  LIN {X 12250.007,Y 1961.237,Z 18.185,A 87.94718,B 0.00000,C 180.00000} ; preinsert
  LIN {X 12250.007,Y 1961.237,Z -231.815,A 87.94718,B 0.00000,C 180.00000} ; insert
  LIN {X 12250.007,Y 1961.237,Z -231.815,A 87.94718,B 0.00000,C 180.00000} ; release
  LIN {X 12250.007,Y 1961.237,Z 68.185,A 87.94718,B 0.00000,C 180.00000} ; retreat
  ; Step 908, bar 2215
  LIN {X 12850.007,Y 1961.237,Z 950.053,A 87.94718,B 0.00000,C 180.00000} ; outside
  LIN {X 12850.007,Y 1961.237,Z 18.185,A 87.94718,B 0.00000,C 180.00000} ; preinsert
  LIN {X 12850.007,Y 1961.237,Z -231.815,A 87.94718,B 0.00000,C 180.00000} ; insert
  LIN {X 12850.007,Y 1961.237,Z -231.815,A 87.94718,B 0.00000,C 180.00000} ; release
  LIN {X 12850.007,Y 1961.237,Z 68.185,A 87.94718,B 0.00000,C 180.00000} ; retreat
  ; Step 909, bar 2221
  LIN {X 13450.007,Y 1961.237,Z 950.053,A 87.94718,B 0.00000,C 180.00000} ; outside
  LIN {X 13450.007,Y 1961.237,Z 18.185,A 87.94718,B 0.00000,C 180.00000} ; preinsert
  LIN {X 13450.007,Y 1961.237,Z -231.815,A 87.94718,B 0.00000,C 180.00000} ; insert
  LIN {X 13450.007,Y 1961.237,Z -231.815,A 87.94718,B 0.00000,C 180.00000} ; release
  LIN {X 13450.007,Y 1961.237,Z 68.185,A 87.94718,B 0.00000,C 180.00000} ; retreat
  ; Step 910, bar 2227
  LIN {X 14050.007,Y 1961.237,Z 950.053,A 87.94718,B 0.00000,C 180.00000} ; outside
  LIN {X 14050.007,Y 1961.237,Z 18.185,A 87.94718,B 0.00000,C 180.00000} ; preinsert
  LIN {X 14050.007,Y 1961.237,Z -231.815,A 87.94718,B 0.00000,C 180.00000} ; insert
  LIN {X 14050.007,Y 1961.237,Z -231.815,A 87.94718,B 0.00000,C 180.00000} ; release
  LIN {X 14050.007,Y 1961.237,Z 68.185,A 87.94718,B 0.00000,C 180.00000} ; retreat
  ; Step 911, bar 2233
  LIN {X 14650.007,Y 1961.237,Z 950.053,A 87.94718,B 0.00000,C 180.00000} ; outside
  LIN {X 14650.007,Y 1961.237,Z 18.185,A 87.94718,B 0.00000,C 180.00000} ; preinsert
  LIN {X 14650.007,Y 1961.237,Z -231.815,A 87.94718,B 0.00000,C 180.00000} ; insert
  LIN {X 14650.007,Y 1961.237,Z -231.815,A 87.94718,B 0.00000,C 180.00000} ; release
  LIN {X 14650.007,Y 1961.237,Z 68.185,A 87.94718,B 0.00000,C 180.00000} ; retreat
  ; Step 912, bar 2239
  LIN {X 15250.007,Y 1961.237,Z 950.053,A 87.94718,B 0.00000,C 180.00000} ; outside
  LIN {X 15250.007,Y 1961.237,Z 18.185,A 87.94718,B 0.00000,C 180.00000} ; preinsert
  LIN {X 15250.007,Y 1961.237,Z -231.815,A 87.94718,B 0.00000,C 180.00000} ; insert
  LIN {X 15250.007,Y 1961.237,Z -231.815,A 87.94718,B 0.00000,C 180.00000} ; release
  LIN {X 15250.007,Y 1961.237,Z 68.185,A 87.94718,B 0.00000,C 180.00000} ; retreat
  ; Step 913, bar 2245
  LIN {X 15850.007,Y 1961.237,Z 950.053,A 87.94718,B 0.00000,C 180.00000} ; outside
  LIN {X 15850.007,Y 1961.237,Z 18.185,A 87.94718,B 0.00000,C 180.00000} ; preinsert
  LIN {X 15850.007,Y 1961.237,Z -231.815,A 87.94718,B 0.00000,C 180.00000} ; insert
  LIN {X 15850.007,Y 1961.237,Z -231.815,A 87.94718,B 0.00000,C 180.00000} ; release
  LIN {X 15850.007,Y 1961.237,Z 68.185,A 87.94718,B 0.00000,C 180.00000} ; retreat
  ; Step 914, bar 298
  LIN {X 0.000,Y -2740.000,Z 1104.371,A 0.00000,B 0.00000,C 180.00000} ; outside
  LIN {X 0.000,Y -2740.000,Z 176.496,A 0.00000,B 0.00000,C 180.00000} ; preinsert
  LIN {X 0.000,Y -2740.000,Z -73.504,A 0.00000,B 0.00000,C 180.00000} ; insert
  LIN {X 0.000,Y -2740.000,Z -73.504,A 0.00000,B 0.00000,C 180.00000} ; release
  LIN {X 0.000,Y -2740.000,Z 226.496,A 0.00000,B 0.00000,C 180.00000} ; retreat
  ; Step 915, bar 325
  LIN {X 0.000,Y 2740.000,Z 1104.371,A 0.00000,B 0.00000,C 180.00000} ; outside
  LIN {X 0.000,Y 2740.000,Z 176.496,A 0.00000,B 0.00000,C 180.00000} ; preinsert
  LIN {X 0.000,Y 2740.000,Z -73.504,A 0.00000,B 0.00000,C 180.00000} ; insert
  LIN {X 0.000,Y 2740.000,Z -73.504,A 0.00000,B 0.00000,C 180.00000} ; release
  LIN {X 0.000,Y 2740.000,Z 226.496,A 0.00000,B 0.00000,C 180.00000} ; retreat
  ; Step 916, bar 284
  LIN {X 0.000,Y -750.000,Z 1108.746,A 0.00000,B 0.00000,C 180.00000} ; outside
  LIN {X 0.000,Y -750.000,Z 178.683,A 0.00000,B 0.00000,C 180.00000} ; preinsert
  LIN {X 0.000,Y -750.000,Z -71.317,A 0.00000,B 0.00000,C 180.00000} ; insert
  LIN {X 0.000,Y -750.000,Z -71.317,A 0.00000,B 0.00000,C 180.00000} ; release
  LIN {X 0.000,Y -750.000,Z 228.683,A 0.00000,B 0.00000,C 180.00000} ; retreat
  ; Step 917, bar 311
  LIN {X 0.000,Y 750.000,Z 1108.746,A 0.00000,B 0.00000,C 180.00000} ; outside
  LIN {X 0.000,Y 750.000,Z 178.683,A 0.00000,B 0.00000,C 180.00000} ; preinsert
  LIN {X 0.000,Y 750.000,Z -71.317,A 0.00000,B 0.00000,C 180.00000} ; insert
  LIN {X 0.000,Y 750.000,Z -71.317,A 0.00000,B 0.00000,C 180.00000} ; release
  LIN {X 0.000,Y 750.000,Z 228.683,A 0.00000,B 0.00000,C 180.00000} ; retreat
  ; Step 918, bar 3105
  LIN {X -15204.133,Y -641.217,Z 1079.276,A -179.87076,B 0.00000,C 180.00000} ; outside
  LIN {X -15204.133,Y -641.217,Z 104.517,A -179.87076,B 0.00000,C 180.00000} ; preinsert
  LIN {X -15204.133,Y -641.217,Z -145.483,A -179.87076,B 0.00000,C 180.00000} ; insert
  LIN {X -15204.133,Y -641.217,Z -145.483,A -179.87076,B 0.00000,C 180.00000} ; release
  LIN {X -15204.133,Y -641.217,Z 154.517,A -179.87076,B 0.00000,C 180.00000} ; retreat
  ; Step 919, bar 3095
  LIN {X 15204.133,Y -641.217,Z 1079.276,A -0.12924,B 0.00000,C 180.00000} ; outside
  LIN {X 15204.133,Y -641.217,Z 104.517,A -0.12924,B 0.00000,C 180.00000} ; preinsert
  LIN {X 15204.133,Y -641.217,Z -145.483,A -0.12924,B 0.00000,C 180.00000} ; insert
  LIN {X 15204.133,Y -641.217,Z -145.483,A -0.12924,B 0.00000,C 180.00000} ; release
  LIN {X 15204.133,Y -641.217,Z 154.517,A -0.12924,B 0.00000,C 180.00000} ; retreat
  ; Step 920, bar 3100
  LIN {X -15204.133,Y 641.217,Z 1079.276,A 179.87076,B 0.00000,C 180.00000} ; outside
  LIN {X -15204.133,Y 641.217,Z 104.517,A 179.87076,B 0.00000,C 180.00000} ; preinsert
  LIN {X -15204.133,Y 641.217,Z -145.483,A 179.87076,B 0.00000,C 180.00000} ; insert
  LIN {X -15204.133,Y 641.217,Z -145.483,A 179.87076,B 0.00000,C 180.00000} ; release
  LIN {X -15204.133,Y 641.217,Z 154.517,A 179.87076,B 0.00000,C 180.00000} ; retreat
  ; Step 921, bar 3090
  LIN {X 15204.133,Y 641.217,Z 1079.276,A 0.12924,B 0.00000,C 180.00000} ; outside
  LIN {X 15204.133,Y 641.217,Z 104.517,A 0.12924,B 0.00000,C 180.00000} ; preinsert
  LIN {X 15204.133,Y 641.217,Z -145.483,A 0.12924,B 0.00000,C 180.00000} ; insert
  LIN {X 15204.133,Y 641.217,Z -145.483,A 0.12924,B 0.00000,C 180.00000} ; release
  LIN {X 15204.133,Y 641.217,Z 154.517,A 0.12924,B 0.00000,C 180.00000} ; retreat
  ; Step 922, bar 2755
  LIN {X -1500.007,Y -1396.237,Z 955.597,A -92.05282,B 0.00000,C -180.00000} ; outside
  LIN {X -1500.007,Y -1396.237,Z 24.092,A -92.05282,B 0.00000,C -180.00000} ; preinsert
  LIN {X -1500.007,Y -1396.237,Z -225.908,A -92.05282,B 0.00000,C -180.00000} ; insert
  LIN {X -1500.007,Y -1396.237,Z -225.908,A -92.05282,B 0.00000,C -180.00000} ; release
  LIN {X -1500.007,Y -1396.237,Z 74.092,A -92.05282,B 0.00000,C -180.00000} ; retreat
  ; Step 923, bar 2752
  LIN {X -750.007,Y -1396.237,Z 955.597,A -92.05282,B 0.00000,C -180.00000} ; outside
  LIN {X -750.007,Y -1396.237,Z 24.092,A -92.05282,B 0.00000,C -180.00000} ; preinsert
  LIN {X -750.007,Y -1396.237,Z -225.908,A -92.05282,B 0.00000,C -180.00000} ; insert
  LIN {X -750.007,Y -1396.237,Z -225.908,A -92.05282,B 0.00000,C -180.00000} ; release
  LIN {X -750.007,Y -1396.237,Z 74.092,A -92.05282,B 0.00000,C -180.00000} ; retreat
  ; Step 924, bar 2749
  LIN {X -0.007,Y -1396.237,Z 955.597,A -92.05282,B 0.00000,C -180.00000} ; outside
  LIN {X -0.007,Y -1396.237,Z 24.092,A -92.05282,B 0.00000,C -180.00000} ; preinsert
  LIN {X -0.007,Y -1396.237,Z -225.908,A -92.05282,B 0.00000,C -180.00000} ; insert
  LIN {X -0.007,Y -1396.237,Z -225.908,A -92.05282,B 0.00000,C -180.00000} ; release
  LIN {X -0.007,Y -1396.237,Z 74.092,A -92.05282,B 0.00000,C -180.00000} ; retreat
  ; Step 925, bar 2758
  LIN {X -2250.007,Y -1396.237,Z 955.597,A -92.05282,B 0.00000,C -180.00000} ; outside
  LIN {X -2250.007,Y -1396.237,Z 24.092,A -92.05282,B 0.00000,C -180.00000} ; preinsert
  LIN {X -2250.007,Y -1396.237,Z -225.908,A -92.05282,B 0.00000,C -180.00000} ; insert
  LIN {X -2250.007,Y -1396.237,Z -225.908,A -92.05282,B 0.00000,C -180.00000} ; release
  LIN {X -2250.007,Y -1396.237,Z 74.092,A -92.05282,B 0.00000,C -180.00000} ; retreat
  ; Step 926, bar 2761
  LIN {X -3000.007,Y -1396.237,Z 955.597,A -92.05282,B 0.00000,C -180.00000} ; outside
  LIN {X -3000.007,Y -1396.237,Z 24.092,A -92.05282,B 0.00000,C -180.00000} ; preinsert
  LIN {X -3000.007,Y -1396.237,Z -225.908,A -92.05282,B 0.00000,C -180.00000} ; insert
  LIN {X -3000.007,Y -1396.237,Z -225.908,A -92.05282,B 0.00000,C -180.00000} ; release
  LIN {X -3000.007,Y -1396.237,Z 74.092,A -92.05282,B 0.00000,C -180.00000} ; retreat
  ; Step 927, bar 2764
  LIN {X -3750.007,Y -1396.237,Z 955.597,A -92.05282,B 0.00000,C -180.00000} ; outside
  LIN {X -3750.007,Y -1396.237,Z 24.092,A -92.05282,B 0.00000,C -180.00000} ; preinsert
  LIN {X -3750.007,Y -1396.237,Z -225.908,A -92.05282,B 0.00000,C -180.00000} ; insert
  LIN {X -3750.007,Y -1396.237,Z -225.908,A -92.05282,B 0.00000,C -180.00000} ; release
  LIN {X -3750.007,Y -1396.237,Z 74.092,A -92.05282,B 0.00000,C -180.00000} ; retreat
  ; Step 928, bar 2767
  LIN {X -4500.007,Y -1396.237,Z 955.597,A -92.05282,B 0.00000,C -180.00000} ; outside
  LIN {X -4500.007,Y -1396.237,Z 24.092,A -92.05282,B 0.00000,C -180.00000} ; preinsert
  LIN {X -4500.007,Y -1396.237,Z -225.908,A -92.05282,B 0.00000,C -180.00000} ; insert
  LIN {X -4500.007,Y -1396.237,Z -225.908,A -92.05282,B 0.00000,C -180.00000} ; release
  LIN {X -4500.007,Y -1396.237,Z 74.092,A -92.05282,B 0.00000,C -180.00000} ; retreat
  ; Step 929, bar 2770
  LIN {X -5250.007,Y -1396.237,Z 955.597,A -92.05282,B 0.00000,C -180.00000} ; outside
  LIN {X -5250.007,Y -1396.237,Z 24.092,A -92.05282,B 0.00000,C -180.00000} ; preinsert
  LIN {X -5250.007,Y -1396.237,Z -225.908,A -92.05282,B 0.00000,C -180.00000} ; insert
  LIN {X -5250.007,Y -1396.237,Z -225.908,A -92.05282,B 0.00000,C -180.00000} ; release
  LIN {X -5250.007,Y -1396.237,Z 74.092,A -92.05282,B 0.00000,C -180.00000} ; retreat
  ; Step 930, bar 2773
  LIN {X -6000.007,Y -1396.237,Z 955.597,A -92.05282,B 0.00000,C -180.00000} ; outside
  LIN {X -6000.007,Y -1396.237,Z 24.092,A -92.05282,B 0.00000,C -180.00000} ; preinsert
  LIN {X -6000.007,Y -1396.237,Z -225.908,A -92.05282,B 0.00000,C -180.00000} ; insert
  LIN {X -6000.007,Y -1396.237,Z -225.908,A -92.05282,B 0.00000,C -180.00000} ; release
  LIN {X -6000.007,Y -1396.237,Z 74.092,A -92.05282,B 0.00000,C -180.00000} ; retreat
  ; Step 931, bar 2776
  LIN {X -6750.007,Y -1396.237,Z 955.597,A -92.05282,B 0.00000,C -180.00000} ; outside
  LIN {X -6750.007,Y -1396.237,Z 24.092,A -92.05282,B 0.00000,C -180.00000} ; preinsert
  LIN {X -6750.007,Y -1396.237,Z -225.908,A -92.05282,B 0.00000,C -180.00000} ; insert
  LIN {X -6750.007,Y -1396.237,Z -225.908,A -92.05282,B 0.00000,C -180.00000} ; release
  LIN {X -6750.007,Y -1396.237,Z 74.092,A -92.05282,B 0.00000,C -180.00000} ; retreat
  ; Step 932, bar 2779
  LIN {X -7500.007,Y -1396.237,Z 955.597,A -92.05282,B 0.00000,C -180.00000} ; outside
  LIN {X -7500.007,Y -1396.237,Z 24.092,A -92.05282,B 0.00000,C -180.00000} ; preinsert
  LIN {X -7500.007,Y -1396.237,Z -225.908,A -92.05282,B 0.00000,C -180.00000} ; insert
  LIN {X -7500.007,Y -1396.237,Z -225.908,A -92.05282,B 0.00000,C -180.00000} ; release
  LIN {X -7500.007,Y -1396.237,Z 74.092,A -92.05282,B 0.00000,C -180.00000} ; retreat
  ; Step 933, bar 2782
  LIN {X -8250.007,Y -1396.237,Z 955.597,A -92.05282,B 0.00000,C -180.00000} ; outside
  LIN {X -8250.007,Y -1396.237,Z 24.092,A -92.05282,B 0.00000,C -180.00000} ; preinsert
  LIN {X -8250.007,Y -1396.237,Z -225.908,A -92.05282,B 0.00000,C -180.00000} ; insert
  LIN {X -8250.007,Y -1396.237,Z -225.908,A -92.05282,B 0.00000,C -180.00000} ; release
  LIN {X -8250.007,Y -1396.237,Z 74.092,A -92.05282,B 0.00000,C -180.00000} ; retreat
  ; Step 934, bar 2785
  LIN {X -9000.007,Y -1396.237,Z 955.597,A -92.05282,B 0.00000,C -180.00000} ; outside
  LIN {X -9000.007,Y -1396.237,Z 24.092,A -92.05282,B 0.00000,C -180.00000} ; preinsert
  LIN {X -9000.007,Y -1396.237,Z -225.908,A -92.05282,B 0.00000,C -180.00000} ; insert
  LIN {X -9000.007,Y -1396.237,Z -225.908,A -92.05282,B 0.00000,C -180.00000} ; release
  LIN {X -9000.007,Y -1396.237,Z 74.092,A -92.05282,B 0.00000,C -180.00000} ; retreat
  ; Step 935, bar 2788
  LIN {X -9750.007,Y -1396.237,Z 955.597,A -92.05282,B 0.00000,C -180.00000} ; outside
  LIN {X -9750.007,Y -1396.237,Z 24.092,A -92.05282,B 0.00000,C -180.00000} ; preinsert
  LIN {X -9750.007,Y -1396.237,Z -225.908,A -92.05282,B 0.00000,C -180.00000} ; insert
  LIN {X -9750.007,Y -1396.237,Z -225.908,A -92.05282,B 0.00000,C -180.00000} ; release
  LIN {X -9750.007,Y -1396.237,Z 74.092,A -92.05282,B 0.00000,C -180.00000} ; retreat
  ; Step 936, bar 2791
  LIN {X -10500.007,Y -1396.237,Z 955.597,A -92.05282,B 0.00000,C -180.00000} ; outside
  LIN {X -10500.007,Y -1396.237,Z 24.092,A -92.05282,B 0.00000,C -180.00000} ; preinsert
  LIN {X -10500.007,Y -1396.237,Z -225.908,A -92.05282,B 0.00000,C -180.00000} ; insert
  LIN {X -10500.007,Y -1396.237,Z -225.908,A -92.05282,B 0.00000,C -180.00000} ; release
  LIN {X -10500.007,Y -1396.237,Z 74.092,A -92.05282,B 0.00000,C -180.00000} ; retreat
  ; Step 937, bar 2794
  LIN {X -11250.007,Y -1396.237,Z 955.597,A -92.05282,B 0.00000,C -180.00000} ; outside
  LIN {X -11250.007,Y -1396.237,Z 24.092,A -92.05282,B 0.00000,C -180.00000} ; preinsert
  LIN {X -11250.007,Y -1396.237,Z -225.908,A -92.05282,B 0.00000,C -180.00000} ; insert
  LIN {X -11250.007,Y -1396.237,Z -225.908,A -92.05282,B 0.00000,C -180.00000} ; release
  LIN {X -11250.007,Y -1396.237,Z 74.092,A -92.05282,B 0.00000,C -180.00000} ; retreat
  ; Step 938, bar 2797
  LIN {X -12000.007,Y -1396.237,Z 955.597,A -92.05282,B 0.00000,C -180.00000} ; outside
  LIN {X -12000.007,Y -1396.237,Z 24.092,A -92.05282,B 0.00000,C -180.00000} ; preinsert
  LIN {X -12000.007,Y -1396.237,Z -225.908,A -92.05282,B 0.00000,C -180.00000} ; insert
  LIN {X -12000.007,Y -1396.237,Z -225.908,A -92.05282,B 0.00000,C -180.00000} ; release
  LIN {X -12000.007,Y -1396.237,Z 74.092,A -92.05282,B 0.00000,C -180.00000} ; retreat
  ; Step 939, bar 2638
  LIN {X 750.007,Y 1396.237,Z 955.597,A 87.94718,B 0.00000,C 180.00000} ; outside
  LIN {X 750.007,Y 1396.237,Z 24.092,A 87.94718,B 0.00000,C 180.00000} ; preinsert
  LIN {X 750.007,Y 1396.237,Z -225.908,A 87.94718,B 0.00000,C 180.00000} ; insert
  LIN {X 750.007,Y 1396.237,Z -225.908,A 87.94718,B 0.00000,C 180.00000} ; release
  LIN {X 750.007,Y 1396.237,Z 74.092,A 87.94718,B 0.00000,C 180.00000} ; retreat
  ; Step 940, bar 2641
  LIN {X 1500.007,Y 1396.237,Z 955.597,A 87.94718,B 0.00000,C -180.00000} ; outside
  LIN {X 1500.007,Y 1396.237,Z 24.092,A 87.94718,B 0.00000,C -180.00000} ; preinsert
  LIN {X 1500.007,Y 1396.237,Z -225.908,A 87.94718,B 0.00000,C -180.00000} ; insert
  LIN {X 1500.007,Y 1396.237,Z -225.908,A 87.94718,B 0.00000,C -180.00000} ; release
  LIN {X 1500.007,Y 1396.237,Z 74.092,A 87.94718,B 0.00000,C -180.00000} ; retreat
  ; Step 941, bar 2644
  LIN {X 2250.007,Y 1396.237,Z 955.597,A 87.94718,B 0.00000,C -180.00000} ; outside
  LIN {X 2250.007,Y 1396.237,Z 24.092,A 87.94718,B 0.00000,C -180.00000} ; preinsert
  LIN {X 2250.007,Y 1396.237,Z -225.908,A 87.94718,B 0.00000,C -180.00000} ; insert
  LIN {X 2250.007,Y 1396.237,Z -225.908,A 87.94718,B 0.00000,C -180.00000} ; release
  LIN {X 2250.007,Y 1396.237,Z 74.092,A 87.94718,B 0.00000,C -180.00000} ; retreat
  ; Step 942, bar 2647
  LIN {X 3000.007,Y 1396.237,Z 955.597,A 87.94718,B 0.00000,C -180.00000} ; outside
  LIN {X 3000.007,Y 1396.237,Z 24.092,A 87.94718,B 0.00000,C -180.00000} ; preinsert
  LIN {X 3000.007,Y 1396.237,Z -225.908,A 87.94718,B 0.00000,C -180.00000} ; insert
  LIN {X 3000.007,Y 1396.237,Z -225.908,A 87.94718,B 0.00000,C -180.00000} ; release
  LIN {X 3000.007,Y 1396.237,Z 74.092,A 87.94718,B 0.00000,C -180.00000} ; retreat
  ; Step 943, bar 2650
  LIN {X 3750.007,Y 1396.237,Z 955.597,A 87.94718,B 0.00000,C -180.00000} ; outside
  LIN {X 3750.007,Y 1396.237,Z 24.092,A 87.94718,B 0.00000,C -180.00000} ; preinsert
  LIN {X 3750.007,Y 1396.237,Z -225.908,A 87.94718,B 0.00000,C -180.00000} ; insert
  LIN {X 3750.007,Y 1396.237,Z -225.908,A 87.94718,B 0.00000,C -180.00000} ; release
  LIN {X 3750.007,Y 1396.237,Z 74.092,A 87.94718,B 0.00000,C -180.00000} ; retreat
  ; Step 944, bar 2653
  LIN {X 4500.007,Y 1396.237,Z 955.597,A 87.94718,B 0.00000,C 180.00000} ; outside
  LIN {X 4500.007,Y 1396.237,Z 24.092,A 87.94718,B 0.00000,C 180.00000} ; preinsert
  LIN {X 4500.007,Y 1396.237,Z -225.908,A 87.94718,B 0.00000,C 180.00000} ; insert
  LIN {X 4500.007,Y 1396.237,Z -225.908,A 87.94718,B 0.00000,C 180.00000} ; release
  LIN {X 4500.007,Y 1396.237,Z 74.092,A 87.94718,B 0.00000,C 180.00000} ; retreat
  ; Step 945, bar 2656
  LIN {X 5250.007,Y 1396.237,Z 955.597,A 87.94718,B 0.00000,C 180.00000} ; outside
  LIN {X 5250.007,Y 1396.237,Z 24.092,A 87.94718,B 0.00000,C 180.00000} ; preinsert
  LIN {X 5250.007,Y 1396.237,Z -225.908,A 87.94718,B 0.00000,C 180.00000} ; insert
  LIN {X 5250.007,Y 1396.237,Z -225.908,A 87.94718,B 0.00000,C 180.00000} ; release
  LIN {X 5250.007,Y 1396.237,Z 74.092,A 87.94718,B 0.00000,C 180.00000} ; retreat
  ; Step 946, bar 2659
  LIN {X 6000.007,Y 1396.237,Z 955.597,A 87.94718,B 0.00000,C 180.00000} ; outside
  LIN {X 6000.007,Y 1396.237,Z 24.092,A 87.94718,B 0.00000,C 180.00000} ; preinsert
  LIN {X 6000.007,Y 1396.237,Z -225.908,A 87.94718,B 0.00000,C 180.00000} ; insert
  LIN {X 6000.007,Y 1396.237,Z -225.908,A 87.94718,B 0.00000,C 180.00000} ; release
  LIN {X 6000.007,Y 1396.237,Z 74.092,A 87.94718,B 0.00000,C 180.00000} ; retreat
  ; Step 947, bar 2662
  LIN {X 6750.007,Y 1396.237,Z 955.597,A 87.94718,B 0.00000,C 180.00000} ; outside
  LIN {X 6750.007,Y 1396.237,Z 24.092,A 87.94718,B 0.00000,C 180.00000} ; preinsert
  LIN {X 6750.007,Y 1396.237,Z -225.908,A 87.94718,B 0.00000,C 180.00000} ; insert
  LIN {X 6750.007,Y 1396.237,Z -225.908,A 87.94718,B 0.00000,C 180.00000} ; release
  LIN {X 6750.007,Y 1396.237,Z 74.092,A 87.94718,B 0.00000,C 180.00000} ; retreat
  ; Step 948, bar 2665
  LIN {X 7500.007,Y 1396.237,Z 955.597,A 87.94718,B 0.00000,C 180.00000} ; outside
  LIN {X 7500.007,Y 1396.237,Z 24.092,A 87.94718,B 0.00000,C 180.00000} ; preinsert
  LIN {X 7500.007,Y 1396.237,Z -225.908,A 87.94718,B 0.00000,C 180.00000} ; insert
  LIN {X 7500.007,Y 1396.237,Z -225.908,A 87.94718,B 0.00000,C 180.00000} ; release
  LIN {X 7500.007,Y 1396.237,Z 74.092,A 87.94718,B 0.00000,C 180.00000} ; retreat
  ; Step 949, bar 2668
  LIN {X 8250.007,Y 1396.237,Z 955.597,A 87.94718,B 0.00000,C 180.00000} ; outside
  LIN {X 8250.007,Y 1396.237,Z 24.092,A 87.94718,B 0.00000,C 180.00000} ; preinsert
  LIN {X 8250.007,Y 1396.237,Z -225.908,A 87.94718,B 0.00000,C 180.00000} ; insert
  LIN {X 8250.007,Y 1396.237,Z -225.908,A 87.94718,B 0.00000,C 180.00000} ; release
  LIN {X 8250.007,Y 1396.237,Z 74.092,A 87.94718,B 0.00000,C 180.00000} ; retreat
  ; Step 950, bar 2671
  LIN {X 9000.007,Y 1396.237,Z 955.597,A 87.94718,B 0.00000,C 180.00000} ; outside
  LIN {X 9000.007,Y 1396.237,Z 24.092,A 87.94718,B 0.00000,C 180.00000} ; preinsert
  LIN {X 9000.007,Y 1396.237,Z -225.908,A 87.94718,B 0.00000,C 180.00000} ; insert
  LIN {X 9000.007,Y 1396.237,Z -225.908,A 87.94718,B 0.00000,C 180.00000} ; release
  LIN {X 9000.007,Y 1396.237,Z 74.092,A 87.94718,B 0.00000,C 180.00000} ; retreat
  ; Step 951, bar 2674
  LIN {X 9750.007,Y 1396.237,Z 955.597,A 87.94718,B 0.00000,C 180.00000} ; outside
  LIN {X 9750.007,Y 1396.237,Z 24.092,A 87.94718,B 0.00000,C 180.00000} ; preinsert
  LIN {X 9750.007,Y 1396.237,Z -225.908,A 87.94718,B 0.00000,C 180.00000} ; insert
  LIN {X 9750.007,Y 1396.237,Z -225.908,A 87.94718,B 0.00000,C 180.00000} ; release
  LIN {X 9750.007,Y 1396.237,Z 74.092,A 87.94718,B 0.00000,C 180.00000} ; retreat
  ; Step 952, bar 2677
  LIN {X 10500.007,Y 1396.237,Z 955.597,A 87.94718,B 0.00000,C 180.00000} ; outside
  LIN {X 10500.007,Y 1396.237,Z 24.092,A 87.94718,B 0.00000,C 180.00000} ; preinsert
  LIN {X 10500.007,Y 1396.237,Z -225.908,A 87.94718,B 0.00000,C 180.00000} ; insert
  LIN {X 10500.007,Y 1396.237,Z -225.908,A 87.94718,B 0.00000,C 180.00000} ; release
  LIN {X 10500.007,Y 1396.237,Z 74.092,A 87.94718,B 0.00000,C 180.00000} ; retreat
  ; Step 953, bar 2680
  LIN {X 11250.007,Y 1396.237,Z 955.597,A 87.94718,B 0.00000,C 180.00000} ; outside
  LIN {X 11250.007,Y 1396.237,Z 24.092,A 87.94718,B 0.00000,C 180.00000} ; preinsert
  LIN {X 11250.007,Y 1396.237,Z -225.908,A 87.94718,B 0.00000,C 180.00000} ; insert
  LIN {X 11250.007,Y 1396.237,Z -225.908,A 87.94718,B 0.00000,C 180.00000} ; release
  LIN {X 11250.007,Y 1396.237,Z 74.092,A 87.94718,B 0.00000,C 180.00000} ; retreat
  ; Step 954, bar 2683
  LIN {X 12000.007,Y 1396.237,Z 955.597,A 87.94718,B 0.00000,C 180.00000} ; outside
  LIN {X 12000.007,Y 1396.237,Z 24.092,A 87.94718,B 0.00000,C 180.00000} ; preinsert
  LIN {X 12000.007,Y 1396.237,Z -225.908,A 87.94718,B 0.00000,C 180.00000} ; insert
  LIN {X 12000.007,Y 1396.237,Z -225.908,A 87.94718,B 0.00000,C 180.00000} ; release
  LIN {X 12000.007,Y 1396.237,Z 74.092,A 87.94718,B 0.00000,C 180.00000} ; retreat
  ; Step 955, bar 2800
  LIN {X 750.007,Y -1396.237,Z 955.597,A -87.94718,B 0.00000,C 180.00000} ; outside
  LIN {X 750.007,Y -1396.237,Z 24.092,A -87.94718,B 0.00000,C 180.00000} ; preinsert
  LIN {X 750.007,Y -1396.237,Z -225.908,A -87.94718,B 0.00000,C 180.00000} ; insert
  LIN {X 750.007,Y -1396.237,Z -225.908,A -87.94718,B 0.00000,C 180.00000} ; release
  LIN {X 750.007,Y -1396.237,Z 74.092,A -87.94718,B 0.00000,C 180.00000} ; retreat
  ; Step 956, bar 2803
  LIN {X 1500.007,Y -1396.237,Z 955.597,A -87.94718,B 0.00000,C -180.00000} ; outside
  LIN {X 1500.007,Y -1396.237,Z 24.092,A -87.94718,B 0.00000,C -180.00000} ; preinsert
  LIN {X 1500.007,Y -1396.237,Z -225.908,A -87.94718,B 0.00000,C -180.00000} ; insert
  LIN {X 1500.007,Y -1396.237,Z -225.908,A -87.94718,B 0.00000,C -180.00000} ; release
  LIN {X 1500.007,Y -1396.237,Z 74.092,A -87.94718,B 0.00000,C -180.00000} ; retreat
  ; Step 957, bar 2806
  LIN {X 2250.007,Y -1396.237,Z 955.597,A -87.94718,B 0.00000,C -180.00000} ; outside
  LIN {X 2250.007,Y -1396.237,Z 24.092,A -87.94718,B 0.00000,C -180.00000} ; preinsert
  LIN {X 2250.007,Y -1396.237,Z -225.908,A -87.94718,B 0.00000,C -180.00000} ; insert
  LIN {X 2250.007,Y -1396.237,Z -225.908,A -87.94718,B 0.00000,C -180.00000} ; release
  LIN {X 2250.007,Y -1396.237,Z 74.092,A -87.94718,B 0.00000,C -180.00000} ; retreat
  ; Step 958, bar 2809
  LIN {X 3000.007,Y -1396.237,Z 955.597,A -87.94718,B 0.00000,C -180.00000} ; outside
  LIN {X 3000.007,Y -1396.237,Z 24.092,A -87.94718,B 0.00000,C -180.00000} ; preinsert
  LIN {X 3000.007,Y -1396.237,Z -225.908,A -87.94718,B 0.00000,C -180.00000} ; insert
  LIN {X 3000.007,Y -1396.237,Z -225.908,A -87.94718,B 0.00000,C -180.00000} ; release
  LIN {X 3000.007,Y -1396.237,Z 74.092,A -87.94718,B 0.00000,C -180.00000} ; retreat
  ; Step 959, bar 2812
  LIN {X 3750.007,Y -1396.237,Z 955.597,A -87.94718,B 0.00000,C -180.00000} ; outside
  LIN {X 3750.007,Y -1396.237,Z 24.092,A -87.94718,B 0.00000,C -180.00000} ; preinsert
  LIN {X 3750.007,Y -1396.237,Z -225.908,A -87.94718,B 0.00000,C -180.00000} ; insert
  LIN {X 3750.007,Y -1396.237,Z -225.908,A -87.94718,B 0.00000,C -180.00000} ; release
  LIN {X 3750.007,Y -1396.237,Z 74.092,A -87.94718,B 0.00000,C -180.00000} ; retreat
  ; Step 960, bar 2815
  LIN {X 4500.007,Y -1396.237,Z 955.597,A -87.94718,B 0.00000,C 180.00000} ; outside
  LIN {X 4500.007,Y -1396.237,Z 24.092,A -87.94718,B 0.00000,C 180.00000} ; preinsert
  LIN {X 4500.007,Y -1396.237,Z -225.908,A -87.94718,B 0.00000,C 180.00000} ; insert
  LIN {X 4500.007,Y -1396.237,Z -225.908,A -87.94718,B 0.00000,C 180.00000} ; release
  LIN {X 4500.007,Y -1396.237,Z 74.092,A -87.94718,B 0.00000,C 180.00000} ; retreat
  ; Step 961, bar 2818
  LIN {X 5250.007,Y -1396.237,Z 955.597,A -87.94718,B 0.00000,C 180.00000} ; outside
  LIN {X 5250.007,Y -1396.237,Z 24.092,A -87.94718,B 0.00000,C 180.00000} ; preinsert
  LIN {X 5250.007,Y -1396.237,Z -225.908,A -87.94718,B 0.00000,C 180.00000} ; insert
  LIN {X 5250.007,Y -1396.237,Z -225.908,A -87.94718,B 0.00000,C 180.00000} ; release
  LIN {X 5250.007,Y -1396.237,Z 74.092,A -87.94718,B 0.00000,C 180.00000} ; retreat
  ; Step 962, bar 2821
  LIN {X 6000.007,Y -1396.237,Z 955.597,A -87.94718,B 0.00000,C 180.00000} ; outside
  LIN {X 6000.007,Y -1396.237,Z 24.092,A -87.94718,B 0.00000,C 180.00000} ; preinsert
  LIN {X 6000.007,Y -1396.237,Z -225.908,A -87.94718,B 0.00000,C 180.00000} ; insert
  LIN {X 6000.007,Y -1396.237,Z -225.908,A -87.94718,B 0.00000,C 180.00000} ; release
  LIN {X 6000.007,Y -1396.237,Z 74.092,A -87.94718,B 0.00000,C 180.00000} ; retreat
  ; Step 963, bar 2824
  LIN {X 6750.007,Y -1396.237,Z 955.597,A -87.94718,B 0.00000,C 180.00000} ; outside
  LIN {X 6750.007,Y -1396.237,Z 24.092,A -87.94718,B 0.00000,C 180.00000} ; preinsert
  LIN {X 6750.007,Y -1396.237,Z -225.908,A -87.94718,B 0.00000,C 180.00000} ; insert
  LIN {X 6750.007,Y -1396.237,Z -225.908,A -87.94718,B 0.00000,C 180.00000} ; release
  LIN {X 6750.007,Y -1396.237,Z 74.092,A -87.94718,B 0.00000,C 180.00000} ; retreat
  ; Step 964, bar 2827
  LIN {X 7500.007,Y -1396.237,Z 955.597,A -87.94718,B 0.00000,C 180.00000} ; outside
  LIN {X 7500.007,Y -1396.237,Z 24.092,A -87.94718,B 0.00000,C 180.00000} ; preinsert
  LIN {X 7500.007,Y -1396.237,Z -225.908,A -87.94718,B 0.00000,C 180.00000} ; insert
  LIN {X 7500.007,Y -1396.237,Z -225.908,A -87.94718,B 0.00000,C 180.00000} ; release
  LIN {X 7500.007,Y -1396.237,Z 74.092,A -87.94718,B 0.00000,C 180.00000} ; retreat
  ; Step 965, bar 2830
  LIN {X 8250.007,Y -1396.237,Z 955.597,A -87.94718,B 0.00000,C 180.00000} ; outside
  LIN {X 8250.007,Y -1396.237,Z 24.092,A -87.94718,B 0.00000,C 180.00000} ; preinsert
  LIN {X 8250.007,Y -1396.237,Z -225.908,A -87.94718,B 0.00000,C 180.00000} ; insert
  LIN {X 8250.007,Y -1396.237,Z -225.908,A -87.94718,B 0.00000,C 180.00000} ; release
  LIN {X 8250.007,Y -1396.237,Z 74.092,A -87.94718,B 0.00000,C 180.00000} ; retreat
  ; Step 966, bar 2833
  LIN {X 9000.007,Y -1396.237,Z 955.597,A -87.94718,B 0.00000,C 180.00000} ; outside
  LIN {X 9000.007,Y -1396.237,Z 24.092,A -87.94718,B 0.00000,C 180.00000} ; preinsert
  LIN {X 9000.007,Y -1396.237,Z -225.908,A -87.94718,B 0.00000,C 180.00000} ; insert
  LIN {X 9000.007,Y -1396.237,Z -225.908,A -87.94718,B 0.00000,C 180.00000} ; release
  LIN {X 9000.007,Y -1396.237,Z 74.092,A -87.94718,B 0.00000,C 180.00000} ; retreat
  ; Step 967, bar 2836
  LIN {X 9750.007,Y -1396.237,Z 955.597,A -87.94718,B 0.00000,C 180.00000} ; outside
  LIN {X 9750.007,Y -1396.237,Z 24.092,A -87.94718,B 0.00000,C 180.00000} ; preinsert
  LIN {X 9750.007,Y -1396.237,Z -225.908,A -87.94718,B 0.00000,C 180.00000} ; insert
  LIN {X 9750.007,Y -1396.237,Z -225.908,A -87.94718,B 0.00000,C 180.00000} ; release
  LIN {X 9750.007,Y -1396.237,Z 74.092,A -87.94718,B 0.00000,C 180.00000} ; retreat
  ; Step 968, bar 2839
  LIN {X 10500.007,Y -1396.237,Z 955.597,A -87.94718,B 0.00000,C 180.00000} ; outside
  LIN {X 10500.007,Y -1396.237,Z 24.092,A -87.94718,B 0.00000,C 180.00000} ; preinsert
  LIN {X 10500.007,Y -1396.237,Z -225.908,A -87.94718,B 0.00000,C 180.00000} ; insert
  LIN {X 10500.007,Y -1396.237,Z -225.908,A -87.94718,B 0.00000,C 180.00000} ; release
  LIN {X 10500.007,Y -1396.237,Z 74.092,A -87.94718,B 0.00000,C 180.00000} ; retreat
  ; Step 969, bar 2842
  LIN {X 11250.007,Y -1396.237,Z 955.597,A -87.94718,B 0.00000,C 180.00000} ; outside
  LIN {X 11250.007,Y -1396.237,Z 24.092,A -87.94718,B 0.00000,C 180.00000} ; preinsert
  LIN {X 11250.007,Y -1396.237,Z -225.908,A -87.94718,B 0.00000,C 180.00000} ; insert
  LIN {X 11250.007,Y -1396.237,Z -225.908,A -87.94718,B 0.00000,C 180.00000} ; release
  LIN {X 11250.007,Y -1396.237,Z 74.092,A -87.94718,B 0.00000,C 180.00000} ; retreat
  ; Step 970, bar 2845
  LIN {X 12000.007,Y -1396.237,Z 955.597,A -87.94718,B 0.00000,C 180.00000} ; outside
  LIN {X 12000.007,Y -1396.237,Z 24.092,A -87.94718,B 0.00000,C 180.00000} ; preinsert
  LIN {X 12000.007,Y -1396.237,Z -225.908,A -87.94718,B 0.00000,C 180.00000} ; insert
  LIN {X 12000.007,Y -1396.237,Z -225.908,A -87.94718,B 0.00000,C 180.00000} ; release
  LIN {X 12000.007,Y -1396.237,Z 74.092,A -87.94718,B 0.00000,C 180.00000} ; retreat
  ; Step 971, bar 2633
  LIN {X -12000.007,Y 1396.237,Z 955.597,A 92.05282,B 0.00000,C 180.00000} ; outside
  LIN {X -12000.007,Y 1396.237,Z 24.092,A 92.05282,B 0.00000,C 180.00000} ; preinsert
  LIN {X -12000.007,Y 1396.237,Z -225.908,A 92.05282,B 0.00000,C 180.00000} ; insert
  LIN {X -12000.007,Y 1396.237,Z -225.908,A 92.05282,B 0.00000,C 180.00000} ; release
  LIN {X -12000.007,Y 1396.237,Z 74.092,A 92.05282,B 0.00000,C 180.00000} ; retreat
  ; Step 972, bar 2626
  LIN {X -11250.007,Y 1396.237,Z 955.597,A 92.05282,B 0.00000,C 180.00000} ; outside
  LIN {X -11250.007,Y 1396.237,Z 24.092,A 92.05282,B 0.00000,C 180.00000} ; preinsert
  LIN {X -11250.007,Y 1396.237,Z -225.908,A 92.05282,B 0.00000,C 180.00000} ; insert
  LIN {X -11250.007,Y 1396.237,Z -225.908,A 92.05282,B 0.00000,C 180.00000} ; release
  LIN {X -11250.007,Y 1396.237,Z 74.092,A 92.05282,B 0.00000,C 180.00000} ; retreat
  ; Step 973, bar 2619
  LIN {X -10500.007,Y 1396.237,Z 955.597,A 92.05282,B 0.00000,C 180.00000} ; outside
  LIN {X -10500.007,Y 1396.237,Z 24.092,A 92.05282,B 0.00000,C 180.00000} ; preinsert
  LIN {X -10500.007,Y 1396.237,Z -225.908,A 92.05282,B 0.00000,C 180.00000} ; insert
  LIN {X -10500.007,Y 1396.237,Z -225.908,A 92.05282,B 0.00000,C 180.00000} ; release
  LIN {X -10500.007,Y 1396.237,Z 74.092,A 92.05282,B 0.00000,C 180.00000} ; retreat
  ; Step 974, bar 2612
  LIN {X -9750.007,Y 1396.237,Z 955.597,A 92.05282,B 0.00000,C 180.00000} ; outside
  LIN {X -9750.007,Y 1396.237,Z 24.092,A 92.05282,B 0.00000,C 180.00000} ; preinsert
  LIN {X -9750.007,Y 1396.237,Z -225.908,A 92.05282,B 0.00000,C 180.00000} ; insert
  LIN {X -9750.007,Y 1396.237,Z -225.908,A 92.05282,B 0.00000,C 180.00000} ; release
  LIN {X -9750.007,Y 1396.237,Z 74.092,A 92.05282,B 0.00000,C 180.00000} ; retreat
  ; Step 975, bar 2605
  LIN {X -9000.007,Y 1396.237,Z 955.597,A 92.05282,B 0.00000,C 180.00000} ; outside
  LIN {X -9000.007,Y 1396.237,Z 24.092,A 92.05282,B 0.00000,C 180.00000} ; preinsert
  LIN {X -9000.007,Y 1396.237,Z -225.908,A 92.05282,B 0.00000,C 180.00000} ; insert
  LIN {X -9000.007,Y 1396.237,Z -225.908,A 92.05282,B 0.00000,C 180.00000} ; release
  LIN {X -9000.007,Y 1396.237,Z 74.092,A 92.05282,B 0.00000,C 180.00000} ; retreat
  ; Step 976, bar 2598
  LIN {X -8250.007,Y 1396.237,Z 955.597,A 92.05282,B 0.00000,C 180.00000} ; outside
  LIN {X -8250.007,Y 1396.237,Z 24.092,A 92.05282,B 0.00000,C 180.00000} ; preinsert
  LIN {X -8250.007,Y 1396.237,Z -225.908,A 92.05282,B 0.00000,C 180.00000} ; insert
  LIN {X -8250.007,Y 1396.237,Z -225.908,A 92.05282,B 0.00000,C 180.00000} ; release
  LIN {X -8250.007,Y 1396.237,Z 74.092,A 92.05282,B 0.00000,C 180.00000} ; retreat
  ; Step 977, bar 2591
  LIN {X -7500.007,Y 1396.237,Z 955.597,A 92.05282,B 0.00000,C 180.00000} ; outside
  LIN {X -7500.007,Y 1396.237,Z 24.092,A 92.05282,B 0.00000,C 180.00000} ; preinsert
  LIN {X -7500.007,Y 1396.237,Z -225.908,A 92.05282,B 0.00000,C 180.00000} ; insert
  LIN {X -7500.007,Y 1396.237,Z -225.908,A 92.05282,B 0.00000,C 180.00000} ; release
  LIN {X -7500.007,Y 1396.237,Z 74.092,A 92.05282,B 0.00000,C 180.00000} ; retreat
  ; Step 978, bar 2584
  LIN {X -6750.007,Y 1396.237,Z 955.597,A 92.05282,B 0.00000,C 180.00000} ; outside
  LIN {X -6750.007,Y 1396.237,Z 24.092,A 92.05282,B 0.00000,C 180.00000} ; preinsert
  LIN {X -6750.007,Y 1396.237,Z -225.908,A 92.05282,B 0.00000,C 180.00000} ; insert
  LIN {X -6750.007,Y 1396.237,Z -225.908,A 92.05282,B 0.00000,C 180.00000} ; release
  LIN {X -6750.007,Y 1396.237,Z 74.092,A 92.05282,B 0.00000,C 180.00000} ; retreat
  ; Step 979, bar 2577
  LIN {X -6000.007,Y 1396.237,Z 955.597,A 92.05282,B 0.00000,C 180.00000} ; outside
  LIN {X -6000.007,Y 1396.237,Z 24.092,A 92.05282,B 0.00000,C 180.00000} ; preinsert
  LIN {X -6000.007,Y 1396.237,Z -225.908,A 92.05282,B 0.00000,C 180.00000} ; insert
  LIN {X -6000.007,Y 1396.237,Z -225.908,A 92.05282,B 0.00000,C 180.00000} ; release
  LIN {X -6000.007,Y 1396.237,Z 74.092,A 92.05282,B 0.00000,C 180.00000} ; retreat
  ; Step 980, bar 2570
  LIN {X -5250.007,Y 1396.237,Z 955.597,A 92.05282,B 0.00000,C 180.00000} ; outside
  LIN {X -5250.007,Y 1396.237,Z 24.092,A 92.05282,B 0.00000,C 180.00000} ; preinsert
  LIN {X -5250.007,Y 1396.237,Z -225.908,A 92.05282,B 0.00000,C 180.00000} ; insert
  LIN {X -5250.007,Y 1396.237,Z -225.908,A 92.05282,B 0.00000,C 180.00000} ; release
  LIN {X -5250.007,Y 1396.237,Z 74.092,A 92.05282,B 0.00000,C 180.00000} ; retreat
  ; Step 981, bar 2563
  LIN {X -4500.007,Y 1396.237,Z 955.597,A 92.05282,B 0.00000,C 180.00000} ; outside
  LIN {X -4500.007,Y 1396.237,Z 24.092,A 92.05282,B 0.00000,C 180.00000} ; preinsert
  LIN {X -4500.007,Y 1396.237,Z -225.908,A 92.05282,B 0.00000,C 180.00000} ; insert
  LIN {X -4500.007,Y 1396.237,Z -225.908,A 92.05282,B 0.00000,C 180.00000} ; release
  LIN {X -4500.007,Y 1396.237,Z 74.092,A 92.05282,B 0.00000,C 180.00000} ; retreat
  ; Step 982, bar 2556
  LIN {X -3750.007,Y 1396.237,Z 955.597,A 92.05282,B 0.00000,C 180.00000} ; outside
  LIN {X -3750.007,Y 1396.237,Z 24.092,A 92.05282,B 0.00000,C 180.00000} ; preinsert
  LIN {X -3750.007,Y 1396.237,Z -225.908,A 92.05282,B 0.00000,C 180.00000} ; insert
  LIN {X -3750.007,Y 1396.237,Z -225.908,A 92.05282,B 0.00000,C 180.00000} ; release
  LIN {X -3750.007,Y 1396.237,Z 74.092,A 92.05282,B 0.00000,C 180.00000} ; retreat
  ; Step 983, bar 2549
  LIN {X -3000.007,Y 1396.237,Z 955.597,A 92.05282,B 0.00000,C 180.00000} ; outside
  LIN {X -3000.007,Y 1396.237,Z 24.092,A 92.05282,B 0.00000,C 180.00000} ; preinsert
  LIN {X -3000.007,Y 1396.237,Z -225.908,A 92.05282,B 0.00000,C 180.00000} ; insert
  LIN {X -3000.007,Y 1396.237,Z -225.908,A 92.05282,B 0.00000,C 180.00000} ; release
  LIN {X -3000.007,Y 1396.237,Z 74.092,A 92.05282,B 0.00000,C 180.00000} ; retreat
  ; Step 984, bar 2542
  LIN {X -2250.007,Y 1396.237,Z 955.597,A 92.05282,B 0.00000,C 180.00000} ; outside
  LIN {X -2250.007,Y 1396.237,Z 24.092,A 92.05282,B 0.00000,C 180.00000} ; preinsert
  LIN {X -2250.007,Y 1396.237,Z -225.908,A 92.05282,B 0.00000,C 180.00000} ; insert
  LIN {X -2250.007,Y 1396.237,Z -225.908,A 92.05282,B 0.00000,C 180.00000} ; release
  LIN {X -2250.007,Y 1396.237,Z 74.092,A 92.05282,B 0.00000,C 180.00000} ; retreat
  ; Step 985, bar 2535
  LIN {X -1500.007,Y 1396.237,Z 955.597,A 92.05282,B 0.00000,C 180.00000} ; outside
  LIN {X -1500.007,Y 1396.237,Z 24.092,A 92.05282,B 0.00000,C 180.00000} ; preinsert
  LIN {X -1500.007,Y 1396.237,Z -225.908,A 92.05282,B 0.00000,C 180.00000} ; insert
  LIN {X -1500.007,Y 1396.237,Z -225.908,A 92.05282,B 0.00000,C 180.00000} ; release
  LIN {X -1500.007,Y 1396.237,Z 74.092,A 92.05282,B 0.00000,C 180.00000} ; retreat
  ; Step 986, bar 2528
  LIN {X -750.007,Y 1396.237,Z 955.597,A 92.05282,B 0.00000,C 180.00000} ; outside
  LIN {X -750.007,Y 1396.237,Z 24.092,A 92.05282,B 0.00000,C 180.00000} ; preinsert
  LIN {X -750.007,Y 1396.237,Z -225.908,A 92.05282,B 0.00000,C 180.00000} ; insert
  LIN {X -750.007,Y 1396.237,Z -225.908,A 92.05282,B 0.00000,C 180.00000} ; release
  LIN {X -750.007,Y 1396.237,Z 74.092,A 92.05282,B 0.00000,C 180.00000} ; retreat
  ; Step 987, bar 1969
  LIN {X -0.007,Y 1396.237,Z 955.597,A 92.05282,B 0.00000,C 180.00000} ; outside
  LIN {X -0.007,Y 1396.237,Z 24.092,A 92.05282,B 0.00000,C 180.00000} ; preinsert
  LIN {X -0.007,Y 1396.237,Z -225.908,A 92.05282,B 0.00000,C 180.00000} ; insert
  LIN {X -0.007,Y 1396.237,Z -225.908,A 92.05282,B 0.00000,C 180.00000} ; release
  LIN {X -0.007,Y 1396.237,Z 74.092,A 92.05282,B 0.00000,C 180.00000} ; retreat
  ; Step 988, bar 3108
  LIN {X -12349.947,Y -1484.887,Z 967.977,A -91.75551,B 0.00000,C -180.00000} ; outside
  LIN {X -12349.947,Y -1484.887,Z 37.280,A -91.75551,B 0.00000,C -180.00000} ; preinsert
  LIN {X -12349.947,Y -1484.887,Z -212.720,A -91.75551,B 0.00000,C -180.00000} ; insert
  LIN {X -12349.947,Y -1484.887,Z -212.720,A -91.75551,B 0.00000,C -180.00000} ; release
  LIN {X -12349.947,Y -1484.887,Z 87.280,A -91.75551,B 0.00000,C -180.00000} ; retreat
  ; Step 989, bar 3123
  LIN {X 12349.947,Y 1484.887,Z 967.977,A 88.24449,B 0.00000,C 180.00000} ; outside
  LIN {X 12349.947,Y 1484.887,Z 37.280,A 88.24449,B 0.00000,C 180.00000} ; preinsert
  LIN {X 12349.947,Y 1484.887,Z -212.720,A 88.24449,B 0.00000,C 180.00000} ; insert
  LIN {X 12349.947,Y 1484.887,Z -212.720,A 88.24449,B 0.00000,C 180.00000} ; release
  LIN {X 12349.947,Y 1484.887,Z 87.280,A 88.24449,B 0.00000,C 180.00000} ; retreat
  ; Step 990, bar 3118
  LIN {X 12349.947,Y -1484.887,Z 967.977,A -88.24449,B 0.00000,C 180.00000} ; outside
  LIN {X 12349.947,Y -1484.887,Z 37.280,A -88.24449,B 0.00000,C 180.00000} ; preinsert
  LIN {X 12349.947,Y -1484.887,Z -212.720,A -88.24449,B 0.00000,C 180.00000} ; insert
  LIN {X 12349.947,Y -1484.887,Z -212.720,A -88.24449,B 0.00000,C 180.00000} ; release
  LIN {X 12349.947,Y -1484.887,Z 87.280,A -88.24449,B 0.00000,C 180.00000} ; retreat
  ; Step 991, bar 3113
  LIN {X -12349.947,Y 1484.887,Z 967.977,A 91.75551,B 0.00000,C 180.00000} ; outside
  LIN {X -12349.947,Y 1484.887,Z 37.280,A 91.75551,B 0.00000,C 180.00000} ; preinsert
  LIN {X -12349.947,Y 1484.887,Z -212.720,A 91.75551,B 0.00000,C 180.00000} ; insert
  LIN {X -12349.947,Y 1484.887,Z -212.720,A 91.75551,B 0.00000,C 180.00000} ; release
  LIN {X -12349.947,Y 1484.887,Z 87.280,A 91.75551,B 0.00000,C 180.00000} ; retreat
  ; Step 992, bar 3110
  LIN {X -12749.942,Y -1484.902,Z 976.966,A -91.55051,B 0.00000,C -180.00000} ; outside
  LIN {X -12749.942,Y -1484.902,Z 46.269,A -91.55051,B 0.00000,C -180.00000} ; preinsert
  LIN {X -12749.942,Y -1484.902,Z -203.731,A -91.55051,B 0.00000,C -180.00000} ; insert
  LIN {X -12749.942,Y -1484.902,Z -203.731,A -91.55051,B 0.00000,C -180.00000} ; release
  LIN {X -12749.942,Y -1484.902,Z 96.269,A -91.55051,B 0.00000,C -180.00000} ; retreat
  ; Step 993, bar 3125
  LIN {X 12749.942,Y 1484.902,Z 976.966,A 88.44949,B 0.00000,C 180.00000} ; outside
  LIN {X 12749.942,Y 1484.902,Z 46.269,A 88.44949,B 0.00000,C 180.00000} ; preinsert
  LIN {X 12749.942,Y 1484.902,Z -203.731,A 88.44949,B 0.00000,C 180.00000} ; insert
  LIN {X 12749.942,Y 1484.902,Z -203.731,A 88.44949,B 0.00000,C 180.00000} ; release
  LIN {X 12749.942,Y 1484.902,Z 96.269,A 88.44949,B 0.00000,C 180.00000} ; retreat
  ; Step 994, bar 3120
  LIN {X 12749.942,Y -1484.902,Z 976.966,A -88.44949,B 0.00000,C 180.00000} ; outside
  LIN {X 12749.942,Y -1484.902,Z 46.269,A -88.44949,B 0.00000,C 180.00000} ; preinsert
  LIN {X 12749.942,Y -1484.902,Z -203.731,A -88.44949,B 0.00000,C 180.00000} ; insert
  LIN {X 12749.942,Y -1484.902,Z -203.731,A -88.44949,B 0.00000,C 180.00000} ; release
  LIN {X 12749.942,Y -1484.902,Z 96.269,A -88.44949,B 0.00000,C 180.00000} ; retreat
  ; Step 995, bar 3115
  LIN {X -12749.942,Y 1484.902,Z 976.966,A 91.55051,B 0.00000,C 180.00000} ; outside
  LIN {X -12749.942,Y 1484.902,Z 46.269,A 91.55051,B 0.00000,C 180.00000} ; preinsert
  LIN {X -12749.942,Y 1484.902,Z -203.731,A 91.55051,B 0.00000,C 180.00000} ; insert
  LIN {X -12749.942,Y 1484.902,Z -203.731,A 91.55051,B 0.00000,C 180.00000} ; release
  LIN {X -12749.942,Y 1484.902,Z 96.269,A 91.55051,B 0.00000,C 180.00000} ; retreat
  ; Step 996, bar 3112
  LIN {X -13149.940,Y -1484.852,Z 985.942,A -91.55051,B 0.00000,C 180.00000} ; outside
  LIN {X -13149.940,Y -1484.852,Z 55.245,A -91.55051,B 0.00000,C 180.00000} ; preinsert
  LIN {X -13149.940,Y -1484.852,Z -194.755,A -91.55051,B 0.00000,C 180.00000} ; insert
  LIN {X -13149.940,Y -1484.852,Z -194.755,A -91.55051,B 0.00000,C 180.00000} ; release
  LIN {X -13149.940,Y -1484.852,Z 105.245,A -91.55051,B 0.00000,C 180.00000} ; retreat
  ; Step 997, bar 3127
  LIN {X 13149.940,Y 1484.852,Z 985.942,A 88.44949,B 0.00000,C 180.00000} ; outside
  LIN {X 13149.940,Y 1484.852,Z 55.245,A 88.44949,B 0.00000,C 180.00000} ; preinsert
  LIN {X 13149.940,Y 1484.852,Z -194.755,A 88.44949,B 0.00000,C 180.00000} ; insert
  LIN {X 13149.940,Y 1484.852,Z -194.755,A 88.44949,B 0.00000,C 180.00000} ; release
  LIN {X 13149.940,Y 1484.852,Z 105.245,A 88.44949,B 0.00000,C 180.00000} ; retreat
  ; Step 998, bar 3122
  LIN {X 13149.940,Y -1484.852,Z 985.942,A -88.44949,B 0.00000,C 180.00000} ; outside
  LIN {X 13149.940,Y -1484.852,Z 55.245,A -88.44949,B 0.00000,C 180.00000} ; preinsert
  LIN {X 13149.940,Y -1484.852,Z -194.755,A -88.44949,B 0.00000,C 180.00000} ; insert
  LIN {X 13149.940,Y -1484.852,Z -194.755,A -88.44949,B 0.00000,C 180.00000} ; release
  LIN {X 13149.940,Y -1484.852,Z 105.245,A -88.44949,B 0.00000,C 180.00000} ; retreat
  ; Step 999, bar 3117
  LIN {X -13149.940,Y 1484.852,Z 985.942,A 91.55051,B 0.00000,C -180.00000} ; outside
  LIN {X -13149.940,Y 1484.852,Z 55.245,A 91.55051,B 0.00000,C -180.00000} ; preinsert
  LIN {X -13149.940,Y 1484.852,Z -194.755,A 91.55051,B 0.00000,C -180.00000} ; insert
  LIN {X -13149.940,Y 1484.852,Z -194.755,A 91.55051,B 0.00000,C -180.00000} ; release
  LIN {X -13149.940,Y 1484.852,Z 105.245,A 91.55051,B 0.00000,C -180.00000} ; retreat
  ; Step 1000, bar 3111
  LIN {X -12749.940,Y -1183.154,Z 986.086,A 91.55051,B 0.00000,C -180.00000} ; outside
  LIN {X -12749.940,Y -1183.154,Z 55.390,A 91.55051,B 0.00000,C -180.00000} ; preinsert
  LIN {X -12749.940,Y -1183.154,Z -194.610,A 91.55051,B 0.00000,C -180.00000} ; insert
  LIN {X -12749.940,Y -1183.154,Z -194.610,A 91.55051,B 0.00000,C -180.00000} ; release
  LIN {X -12749.940,Y -1183.154,Z 105.390,A 91.55051,B 0.00000,C -180.00000} ; retreat
  ; Step 1001, bar 3109
  LIN {X -12349.940,Y -1183.154,Z 986.086,A 91.55051,B 0.00000,C -180.00000} ; outside
  LIN {X -12349.940,Y -1183.154,Z 55.390,A 91.55051,B 0.00000,C -180.00000} ; preinsert
  LIN {X -12349.940,Y -1183.154,Z -194.610,A 91.55051,B 0.00000,C -180.00000} ; insert
  LIN {X -12349.940,Y -1183.154,Z -194.610,A 91.55051,B 0.00000,C -180.00000} ; release
  LIN {X -12349.940,Y -1183.154,Z 105.390,A 91.55051,B 0.00000,C -180.00000} ; retreat
  ; Step 1002, bar 3119
  LIN {X 12349.940,Y -1183.154,Z 986.086,A 88.44949,B 0.00000,C 180.00000} ; outside
  LIN {X 12349.940,Y -1183.154,Z 55.390,A 88.44949,B 0.00000,C 180.00000} ; preinsert
  LIN {X 12349.940,Y -1183.154,Z -194.610,A 88.44949,B 0.00000,C 180.00000} ; insert
  LIN {X 12349.940,Y -1183.154,Z -194.610,A 88.44949,B 0.00000,C 180.00000} ; release
  LIN {X 12349.940,Y -1183.154,Z 105.390,A 88.44949,B 0.00000,C 180.00000} ; retreat
  ; Step 1003, bar 3121
  LIN {X 12749.940,Y -1183.154,Z 986.086,A 88.44949,B 0.00000,C 180.00000} ; outside
  LIN {X 12749.940,Y -1183.154,Z 55.390,A 88.44949,B 0.00000,C 180.00000} ; preinsert
  LIN {X 12749.940,Y -1183.154,Z -194.610,A 88.44949,B 0.00000,C 180.00000} ; insert
  LIN {X 12749.940,Y -1183.154,Z -194.610,A 88.44949,B 0.00000,C 180.00000} ; release
  LIN {X 12749.940,Y -1183.154,Z 105.390,A 88.44949,B 0.00000,C 180.00000} ; retreat
  ; Step 1004, bar 3124
  LIN {X 12349.940,Y 1183.154,Z 986.086,A -88.44949,B 0.00000,C 180.00000} ; outside
  LIN {X 12349.940,Y 1183.154,Z 55.390,A -88.44949,B 0.00000,C 180.00000} ; preinsert
  LIN {X 12349.940,Y 1183.154,Z -194.610,A -88.44949,B 0.00000,C 180.00000} ; insert
  LIN {X 12349.940,Y 1183.154,Z -194.610,A -88.44949,B 0.00000,C 180.00000} ; release
  LIN {X 12349.940,Y 1183.154,Z 105.390,A -88.44949,B 0.00000,C 180.00000} ; retreat
  ; Step 1005, bar 3114
  LIN {X -12349.940,Y 1183.154,Z 986.086,A -91.55051,B 0.00000,C 180.00000} ; outside
  LIN {X -12349.940,Y 1183.154,Z 55.390,A -91.55051,B 0.00000,C 180.00000} ; preinsert
  LIN {X -12349.940,Y 1183.154,Z -194.610,A -91.55051,B 0.00000,C 180.00000} ; insert
  LIN {X -12349.940,Y 1183.154,Z -194.610,A -91.55051,B 0.00000,C 180.00000} ; release
  LIN {X -12349.940,Y 1183.154,Z 105.390,A -91.55051,B 0.00000,C 180.00000} ; retreat
  ; Step 1006, bar 3126
  LIN {X 12749.940,Y 1183.154,Z 986.086,A -88.44949,B 0.00000,C 180.00000} ; outside
  LIN {X 12749.940,Y 1183.154,Z 55.390,A -88.44949,B 0.00000,C 180.00000} ; preinsert
  LIN {X 12749.940,Y 1183.154,Z -194.610,A -88.44949,B 0.00000,C 180.00000} ; insert
  LIN {X 12749.940,Y 1183.154,Z -194.610,A -88.44949,B 0.00000,C 180.00000} ; release
  LIN {X 12749.940,Y 1183.154,Z 105.390,A -88.44949,B 0.00000,C 180.00000} ; retreat
  ; Step 1007, bar 3116
  LIN {X -12749.940,Y 1183.154,Z 986.086,A -91.55051,B 0.00000,C 180.00000} ; outside
  LIN {X -12749.940,Y 1183.154,Z 55.390,A -91.55051,B 0.00000,C 180.00000} ; preinsert
  LIN {X -12749.940,Y 1183.154,Z -194.610,A -91.55051,B 0.00000,C 180.00000} ; insert
  LIN {X -12749.940,Y 1183.154,Z -194.610,A -91.55051,B 0.00000,C 180.00000} ; release
  LIN {X -12749.940,Y 1183.154,Z 105.390,A -91.55051,B 0.00000,C 180.00000} ; retreat
  ; Step 1008, bar 299
  LIN {X 0.000,Y -2890.000,Z 1110.621,A 0.00000,B 0.00000,C 180.00000} ; outside
  LIN {X 0.000,Y -2890.000,Z 179.621,A 0.00000,B 0.00000,C 180.00000} ; preinsert
  LIN {X 0.000,Y -2890.000,Z -70.379,A 0.00000,B 0.00000,C 180.00000} ; insert
  LIN {X 0.000,Y -2890.000,Z -70.379,A 0.00000,B 0.00000,C 180.00000} ; release
  LIN {X 0.000,Y -2890.000,Z 229.621,A 0.00000,B 0.00000,C 180.00000} ; retreat
  ; Step 1009, bar 326
  LIN {X 0.000,Y 2890.000,Z 1110.621,A 0.00000,B 0.00000,C 180.00000} ; outside
  LIN {X 0.000,Y 2890.000,Z 179.621,A 0.00000,B 0.00000,C 180.00000} ; preinsert
  LIN {X 0.000,Y 2890.000,Z -70.379,A 0.00000,B 0.00000,C 180.00000} ; insert
  LIN {X 0.000,Y 2890.000,Z -70.379,A 0.00000,B 0.00000,C 180.00000} ; release
  LIN {X 0.000,Y 2890.000,Z 229.621,A 0.00000,B 0.00000,C 180.00000} ; retreat
  ; Step 1010, bar 2975
  LIN {X -14450.007,Y -1026.237,Z 965.399,A -92.05282,B 0.00000,C -180.00000} ; outside
  LIN {X -14450.007,Y -1026.237,Z 32.653,A -92.05282,B 0.00000,C -180.00000} ; preinsert
  LIN {X -14450.007,Y -1026.237,Z -217.347,A -92.05282,B 0.00000,C -180.00000} ; insert
  LIN {X -14450.007,Y -1026.237,Z -217.347,A -92.05282,B 0.00000,C -180.00000} ; release
  LIN {X -14450.007,Y -1026.237,Z 82.653,A -92.05282,B 0.00000,C -180.00000} ; retreat
  ; Step 1011, bar 2995
  LIN {X 14450.007,Y 1026.237,Z 965.399,A 87.94718,B 0.00000,C 180.00000} ; outside
  LIN {X 14450.007,Y 1026.237,Z 32.653,A 87.94718,B 0.00000,C 180.00000} ; preinsert
  LIN {X 14450.007,Y 1026.237,Z -217.347,A 87.94718,B 0.00000,C 180.00000} ; insert
  LIN {X 14450.007,Y 1026.237,Z -217.347,A 87.94718,B 0.00000,C 180.00000} ; release
  LIN {X 14450.007,Y 1026.237,Z 82.653,A 87.94718,B 0.00000,C 180.00000} ; retreat
  ; Step 1012, bar 3014
  LIN {X 14450.007,Y -1026.237,Z 965.399,A -87.94718,B 0.00000,C 180.00000} ; outside
  LIN {X 14450.007,Y -1026.237,Z 32.652,A -87.94718,B 0.00000,C 180.00000} ; preinsert
  LIN {X 14450.007,Y -1026.237,Z -217.348,A -87.94718,B 0.00000,C 180.00000} ; insert
  LIN {X 14450.007,Y -1026.237,Z -217.348,A -87.94718,B 0.00000,C 180.00000} ; release
  LIN {X 14450.007,Y -1026.237,Z 82.652,A -87.94718,B 0.00000,C 180.00000} ; retreat
  ; Step 1013, bar 2956
  LIN {X -14450.007,Y 1026.237,Z 965.399,A 92.05282,B 0.00000,C 180.00000} ; outside
  LIN {X -14450.007,Y 1026.237,Z 32.652,A 92.05282,B 0.00000,C 180.00000} ; preinsert
  LIN {X -14450.007,Y 1026.237,Z -217.348,A 92.05282,B 0.00000,C 180.00000} ; insert
  LIN {X -14450.007,Y 1026.237,Z -217.348,A 92.05282,B 0.00000,C 180.00000} ; release
  LIN {X -14450.007,Y 1026.237,Z 82.652,A 92.05282,B 0.00000,C 180.00000} ; retreat
  ; Step 1014, bar 2970
  LIN {X -13650.059,Y -1026.145,Z 977.187,A 91.75551,B 0.00000,C 180.00000} ; outside
  LIN {X -13650.059,Y -1026.145,Z 44.441,A 91.75551,B 0.00000,C 180.00000} ; preinsert
  LIN {X -13650.059,Y -1026.145,Z -205.559,A 91.75551,B 0.00000,C 180.00000} ; insert
  LIN {X -13650.059,Y -1026.145,Z -205.559,A 91.75551,B 0.00000,C 180.00000} ; release
  LIN {X -13650.059,Y -1026.145,Z 94.441,A 91.75551,B 0.00000,C 180.00000} ; retreat
  ; Step 1015, bar 2989
  LIN {X 13650.059,Y 1026.145,Z 977.187,A -88.24449,B 0.00000,C 180.00000} ; outside
  LIN {X 13650.059,Y 1026.145,Z 44.441,A -88.24449,B 0.00000,C 180.00000} ; preinsert
  LIN {X 13650.059,Y 1026.145,Z -205.559,A -88.24449,B 0.00000,C 180.00000} ; insert
  LIN {X 13650.059,Y 1026.145,Z -205.559,A -88.24449,B 0.00000,C 180.00000} ; release
  LIN {X 13650.059,Y 1026.145,Z 94.441,A -88.24449,B 0.00000,C 180.00000} ; retreat
  ; Step 1016, bar 3009
  LIN {X 13650.059,Y -1026.145,Z 977.187,A 88.24449,B 0.00000,C 180.00000} ; outside
  LIN {X 13650.059,Y -1026.145,Z 44.441,A 88.24449,B 0.00000,C 180.00000} ; preinsert
  LIN {X 13650.059,Y -1026.145,Z -205.559,A 88.24449,B 0.00000,C 180.00000} ; insert
  LIN {X 13650.059,Y -1026.145,Z -205.559,A 88.24449,B 0.00000,C 180.00000} ; release
  LIN {X 13650.059,Y -1026.145,Z 94.441,A 88.24449,B 0.00000,C 180.00000} ; retreat
  ; Step 1017, bar 2950
  LIN {X -13650.059,Y 1026.145,Z 977.187,A -91.75551,B 0.00000,C -180.00000} ; outside
  LIN {X -13650.059,Y 1026.145,Z 44.441,A -91.75551,B 0.00000,C -180.00000} ; preinsert
  LIN {X -13650.059,Y 1026.145,Z -205.559,A -91.75551,B 0.00000,C -180.00000} ; insert
  LIN {X -13650.059,Y 1026.145,Z -205.559,A -91.75551,B 0.00000,C -180.00000} ; release
  LIN {X -13650.059,Y 1026.145,Z 94.441,A -91.75551,B 0.00000,C -180.00000} ; retreat
  ; Step 1018, bar 2965
  LIN {X -12849.916,Y -1026.296,Z 1012.142,A 87.44234,B 0.00000,C -180.00000} ; outside
  LIN {X -12849.916,Y -1026.296,Z 79.396,A 87.44234,B 0.00000,C -180.00000} ; preinsert
  LIN {X -12849.916,Y -1026.296,Z -170.604,A 87.44234,B 0.00000,C -180.00000} ; insert
  LIN {X -12849.916,Y -1026.296,Z -170.604,A 87.44234,B 0.00000,C -180.00000} ; release
  LIN {X -12849.916,Y -1026.296,Z 129.396,A 87.44234,B 0.00000,C -180.00000} ; retreat
  ; Step 1019, bar 3004
  LIN {X 12849.916,Y -1026.296,Z 1012.142,A 92.55766,B 0.00000,C 180.00000} ; outside
  LIN {X 12849.916,Y -1026.296,Z 79.396,A 92.55766,B 0.00000,C 180.00000} ; preinsert
  LIN {X 12849.916,Y -1026.296,Z -170.604,A 92.55766,B 0.00000,C 180.00000} ; insert
  LIN {X 12849.916,Y -1026.296,Z -170.604,A 92.55766,B 0.00000,C 180.00000} ; release
  LIN {X 12849.916,Y -1026.296,Z 129.396,A 92.55766,B 0.00000,C 180.00000} ; retreat
  ; Step 1020, bar 2944
  LIN {X -12849.916,Y 1026.296,Z 1012.142,A -87.44234,B 0.00000,C -180.00000} ; outside
  LIN {X -12849.916,Y 1026.296,Z 79.396,A -87.44234,B 0.00000,C -180.00000} ; preinsert
  LIN {X -12849.916,Y 1026.296,Z -170.604,A -87.44234,B 0.00000,C -180.00000} ; insert
  LIN {X -12849.916,Y 1026.296,Z -170.604,A -87.44234,B 0.00000,C -180.00000} ; release
  LIN {X -12849.916,Y 1026.296,Z 129.396,A -87.44234,B 0.00000,C -180.00000} ; retreat
  ; Step 1021, bar 2983
  LIN {X 12849.916,Y 1026.296,Z 1012.142,A -92.55766,B 0.00000,C -180.00000} ; outside
  LIN {X 12849.916,Y 1026.296,Z 79.396,A -92.55766,B 0.00000,C -180.00000} ; preinsert
  LIN {X 12849.916,Y 1026.296,Z -170.604,A -92.55766,B 0.00000,C -180.00000} ; insert
  LIN {X 12849.916,Y 1026.296,Z -170.604,A -92.55766,B 0.00000,C -180.00000} ; release
  LIN {X 12849.916,Y 1026.296,Z 129.396,A -92.55766,B 0.00000,C -180.00000} ; retreat
  ; Step 1022, bar 283
  LIN {X 0.000,Y -625.000,Z 1113.121,A 0.00000,B 0.00000,C 180.00000} ; outside
  LIN {X 0.000,Y -625.000,Z 180.871,A 0.00000,B 0.00000,C 180.00000} ; preinsert
  LIN {X 0.000,Y -625.000,Z -69.129,A 0.00000,B 0.00000,C 180.00000} ; insert
  LIN {X 0.000,Y -625.000,Z -69.129,A 0.00000,B 0.00000,C 180.00000} ; release
  LIN {X 0.000,Y -625.000,Z 230.871,A 0.00000,B 0.00000,C 180.00000} ; retreat
  ; Step 1023, bar 310
  LIN {X 0.000,Y 625.000,Z 1113.121,A 0.00000,B 0.00000,C 180.00000} ; outside
  LIN {X 0.000,Y 625.000,Z 180.871,A 0.00000,B 0.00000,C 180.00000} ; preinsert
  LIN {X 0.000,Y 625.000,Z -69.129,A 0.00000,B 0.00000,C 180.00000} ; insert
  LIN {X 0.000,Y 625.000,Z -69.129,A 0.00000,B 0.00000,C 180.00000} ; release
  LIN {X 0.000,Y 625.000,Z 230.871,A 0.00000,B 0.00000,C 180.00000} ; retreat
  ; Step 1024, bar 300
  LIN {X 0.000,Y -3040.000,Z 1115.621,A 0.00000,B 0.00000,C 180.00000} ; outside
  LIN {X 0.000,Y -3040.000,Z 182.121,A 0.00000,B 0.00000,C 180.00000} ; preinsert
  LIN {X 0.000,Y -3040.000,Z -67.879,A 0.00000,B 0.00000,C 180.00000} ; insert
  LIN {X 0.000,Y -3040.000,Z -67.879,A 0.00000,B 0.00000,C 180.00000} ; release
  LIN {X 0.000,Y -3040.000,Z 232.121,A 0.00000,B 0.00000,C 180.00000} ; retreat
  ; Step 1025, bar 327
  LIN {X 0.000,Y 3040.000,Z 1115.621,A 0.00000,B 0.00000,C 180.00000} ; outside
  LIN {X 0.000,Y 3040.000,Z 182.121,A 0.00000,B 0.00000,C 180.00000} ; preinsert
  LIN {X 0.000,Y 3040.000,Z -67.879,A 0.00000,B 0.00000,C 180.00000} ; insert
  LIN {X 0.000,Y 3040.000,Z -67.879,A 0.00000,B 0.00000,C 180.00000} ; release
  LIN {X 0.000,Y 3040.000,Z 232.121,A 0.00000,B 0.00000,C 180.00000} ; retreat
  ; Step 1026, bar 282
  LIN {X 0.000,Y -500.000,Z 1118.121,A 0.00000,B 0.00000,C 180.00000} ; outside
  LIN {X 0.000,Y -500.000,Z 183.371,A 0.00000,B 0.00000,C 180.00000} ; preinsert
  LIN {X 0.000,Y -500.000,Z -66.629,A 0.00000,B 0.00000,C 180.00000} ; insert
  LIN {X 0.000,Y -500.000,Z -66.629,A 0.00000,B 0.00000,C 180.00000} ; release
  LIN {X 0.000,Y -500.000,Z 233.371,A 0.00000,B 0.00000,C 180.00000} ; retreat
  ; Step 1027, bar 309
  LIN {X 0.000,Y 500.000,Z 1118.121,A 0.00000,B 0.00000,C 180.00000} ; outside
  LIN {X 0.000,Y 500.000,Z 183.371,A 0.00000,B 0.00000,C 180.00000} ; preinsert
  LIN {X 0.000,Y 500.000,Z -66.629,A 0.00000,B 0.00000,C 180.00000} ; insert
  LIN {X 0.000,Y 500.000,Z -66.629,A 0.00000,B 0.00000,C 180.00000} ; release
  LIN {X 0.000,Y 500.000,Z 233.371,A 0.00000,B 0.00000,C 180.00000} ; retreat
  ; Step 1028, bar 3104
  LIN {X -15204.133,Y -391.217,Z 1079.276,A -179.87076,B 0.00000,C -180.00000} ; outside
  LIN {X -15204.133,Y -391.217,Z 109.830,A -179.87076,B 0.00000,C -180.00000} ; preinsert
  LIN {X -15204.133,Y -391.217,Z -140.170,A -179.87076,B 0.00000,C -180.00000} ; insert
  LIN {X -15204.133,Y -391.217,Z -140.170,A -179.87076,B 0.00000,C -180.00000} ; release
  LIN {X -15204.133,Y -391.217,Z 159.830,A -179.87076,B 0.00000,C -180.00000} ; retreat
  ; Step 1029, bar 3094
  LIN {X 15204.133,Y -391.217,Z 1079.276,A -0.12924,B 0.00000,C 180.00000} ; outside
  LIN {X 15204.133,Y -391.217,Z 109.830,A -0.12924,B 0.00000,C 180.00000} ; preinsert
  LIN {X 15204.133,Y -391.217,Z -140.170,A -0.12924,B 0.00000,C 180.00000} ; insert
  LIN {X 15204.133,Y -391.217,Z -140.170,A -0.12924,B 0.00000,C 180.00000} ; release
  LIN {X 15204.133,Y -391.217,Z 159.830,A -0.12924,B 0.00000,C 180.00000} ; retreat
  ; Step 1030, bar 3099
  LIN {X -15204.133,Y 391.217,Z 1079.276,A 179.87076,B 0.00000,C 180.00000} ; outside
  LIN {X -15204.133,Y 391.217,Z 109.830,A 179.87076,B 0.00000,C 180.00000} ; preinsert
  LIN {X -15204.133,Y 391.217,Z -140.170,A 179.87076,B 0.00000,C 180.00000} ; insert
  LIN {X -15204.133,Y 391.217,Z -140.170,A 179.87076,B 0.00000,C 180.00000} ; release
  LIN {X -15204.133,Y 391.217,Z 159.830,A 179.87076,B 0.00000,C 180.00000} ; retreat
  ; Step 1031, bar 3089
  LIN {X 15204.133,Y 391.217,Z 1079.276,A 0.12924,B 0.00000,C 180.00000} ; outside
  LIN {X 15204.133,Y 391.217,Z 109.830,A 0.12924,B 0.00000,C 180.00000} ; preinsert
  LIN {X 15204.133,Y 391.217,Z -140.170,A 0.12924,B 0.00000,C 180.00000} ; insert
  LIN {X 15204.133,Y 391.217,Z -140.170,A 0.12924,B 0.00000,C 180.00000} ; release
  LIN {X 15204.133,Y 391.217,Z 159.830,A 0.12924,B 0.00000,C 180.00000} ; retreat
  ; Step 1032, bar 301
  LIN {X 0.000,Y -3155.000,Z 1120.922,A 0.00000,B 0.00000,C 180.00000} ; outside
  LIN {X 0.000,Y -3155.000,Z 184.772,A 0.00000,B 0.00000,C 180.00000} ; preinsert
  LIN {X 0.000,Y -3155.000,Z -65.228,A 0.00000,B 0.00000,C 180.00000} ; insert
  LIN {X 0.000,Y -3155.000,Z -65.228,A 0.00000,B 0.00000,C 180.00000} ; release
  LIN {X 0.000,Y -3155.000,Z 234.772,A 0.00000,B 0.00000,C 180.00000} ; retreat
  ; Step 1033, bar 328
  LIN {X 0.000,Y 3155.000,Z 1120.922,A 0.00000,B 0.00000,C 180.00000} ; outside
  LIN {X 0.000,Y 3155.000,Z 184.772,A 0.00000,B 0.00000,C 180.00000} ; preinsert
  LIN {X 0.000,Y 3155.000,Z -65.228,A 0.00000,B 0.00000,C 180.00000} ; insert
  LIN {X 0.000,Y 3155.000,Z -65.228,A 0.00000,B 0.00000,C 180.00000} ; release
  LIN {X 0.000,Y 3155.000,Z 234.772,A 0.00000,B 0.00000,C 180.00000} ; retreat
  ; Step 1034, bar 281
  LIN {X 0.000,Y -375.000,Z 1123.746,A 0.00000,B 0.00000,C 180.00000} ; outside
  LIN {X 0.000,Y -375.000,Z 186.183,A 0.00000,B 0.00000,C 180.00000} ; preinsert
  LIN {X 0.000,Y -375.000,Z -63.817,A 0.00000,B 0.00000,C 180.00000} ; insert
  LIN {X 0.000,Y -375.000,Z -63.817,A 0.00000,B 0.00000,C 180.00000} ; release
  LIN {X 0.000,Y -375.000,Z 236.183,A 0.00000,B 0.00000,C 180.00000} ; retreat
  ; Step 1035, bar 308
  LIN {X 0.000,Y 375.000,Z 1123.746,A 0.00000,B 0.00000,C 180.00000} ; outside
  LIN {X 0.000,Y 375.000,Z 186.183,A 0.00000,B 0.00000,C 180.00000} ; preinsert
  LIN {X 0.000,Y 375.000,Z -63.817,A 0.00000,B 0.00000,C 180.00000} ; insert
  LIN {X 0.000,Y 375.000,Z -63.817,A 0.00000,B 0.00000,C 180.00000} ; release
  LIN {X 0.000,Y 375.000,Z 236.183,A 0.00000,B 0.00000,C 180.00000} ; retreat
  ; Step 1036, bar 3075
  LIN {X 15450.033,Y -1181.101,Z 967.962,A 48.70858,B 0.00000,C 180.00000} ; outside
  LIN {X 15450.033,Y -1181.101,Z 12.331,A 48.70858,B 0.00000,C 180.00000} ; preinsert
  LIN {X 15450.033,Y -1181.101,Z -237.669,A 48.70858,B 0.00000,C 180.00000} ; insert
  LIN {X 15450.033,Y -1181.101,Z -237.669,A 48.70858,B 0.00000,C 180.00000} ; release
  LIN {X 15450.033,Y -1181.101,Z 62.331,A 48.70858,B 0.00000,C 180.00000} ; retreat
  ; Step 1037, bar 3080
  LIN {X 15850.033,Y -1181.101,Z 967.962,A 48.70858,B 0.00000,C 180.00000} ; outside
  LIN {X 15850.033,Y -1181.101,Z 12.331,A 48.70858,B 0.00000,C 180.00000} ; preinsert
  LIN {X 15850.033,Y -1181.101,Z -237.669,A 48.70858,B 0.00000,C 180.00000} ; insert
  LIN {X 15850.033,Y -1181.101,Z -237.669,A 48.70858,B 0.00000,C 180.00000} ; release
  LIN {X 15850.033,Y -1181.101,Z 62.331,A 48.70858,B 0.00000,C 180.00000} ; retreat
  ; Step 1038, bar 3085
  LIN {X 16250.033,Y -1181.101,Z 967.962,A 48.70858,B 0.00000,C 180.00000} ; outside
  LIN {X 16250.033,Y -1181.101,Z 12.331,A 48.70858,B 0.00000,C 180.00000} ; preinsert
  LIN {X 16250.033,Y -1181.101,Z -237.669,A 48.70858,B 0.00000,C 180.00000} ; insert
  LIN {X 16250.033,Y -1181.101,Z -237.669,A 48.70858,B 0.00000,C 180.00000} ; release
  LIN {X 16250.033,Y -1181.101,Z 62.331,A 48.70858,B 0.00000,C 180.00000} ; retreat
  ; Step 1039, bar 3037
  LIN {X -16250.033,Y 1181.101,Z 967.962,A -131.29142,B 0.00000,C -180.00000} ; outside
  LIN {X -16250.033,Y 1181.101,Z 12.331,A -131.29142,B 0.00000,C -180.00000} ; preinsert
  LIN {X -16250.033,Y 1181.101,Z -237.669,A -131.29142,B 0.00000,C -180.00000} ; insert
  LIN {X -16250.033,Y 1181.101,Z -237.669,A -131.29142,B 0.00000,C -180.00000} ; release
  LIN {X -16250.033,Y 1181.101,Z 62.331,A -131.29142,B 0.00000,C -180.00000} ; retreat
  ; Step 1040, bar 3031
  LIN {X -15850.033,Y 1181.101,Z 967.962,A -131.29142,B 0.00000,C -180.00000} ; outside
  LIN {X -15850.033,Y 1181.101,Z 12.331,A -131.29142,B 0.00000,C -180.00000} ; preinsert
  LIN {X -15850.033,Y 1181.101,Z -237.669,A -131.29142,B 0.00000,C -180.00000} ; insert
  LIN {X -15850.033,Y 1181.101,Z -237.669,A -131.29142,B 0.00000,C -180.00000} ; release
  LIN {X -15850.033,Y 1181.101,Z 62.331,A -131.29142,B 0.00000,C -180.00000} ; retreat
  ; Step 1041, bar 3025
  LIN {X -15450.033,Y 1181.101,Z 967.962,A -131.29142,B 0.00000,C -180.00000} ; outside
  LIN {X -15450.033,Y 1181.101,Z 12.331,A -131.29142,B 0.00000,C -180.00000} ; preinsert
  LIN {X -15450.033,Y 1181.101,Z -237.669,A -131.29142,B 0.00000,C -180.00000} ; insert
  LIN {X -15450.033,Y 1181.101,Z -237.669,A -131.29142,B 0.00000,C -180.00000} ; release
  LIN {X -15450.033,Y 1181.101,Z 62.331,A -131.29142,B 0.00000,C -180.00000} ; retreat
  ; Step 1042, bar 3052
  LIN {X -16250.033,Y -1181.101,Z 967.962,A 131.29142,B 0.00000,C 180.00000} ; outside
  LIN {X -16250.033,Y -1181.101,Z 12.331,A 131.29142,B 0.00000,C 180.00000} ; preinsert
  LIN {X -16250.033,Y -1181.101,Z -237.669,A 131.29142,B 0.00000,C 180.00000} ; insert
  LIN {X -16250.033,Y -1181.101,Z -237.669,A 131.29142,B 0.00000,C 180.00000} ; release
  LIN {X -16250.033,Y -1181.101,Z 62.331,A 131.29142,B 0.00000,C 180.00000} ; retreat
  ; Step 1043, bar 3047
  LIN {X -15850.033,Y -1181.101,Z 967.962,A 131.29142,B 0.00000,C 180.00000} ; outside
  LIN {X -15850.033,Y -1181.101,Z 12.331,A 131.29142,B 0.00000,C 180.00000} ; preinsert
  LIN {X -15850.033,Y -1181.101,Z -237.669,A 131.29142,B 0.00000,C 180.00000} ; insert
  LIN {X -15850.033,Y -1181.101,Z -237.669,A 131.29142,B 0.00000,C 180.00000} ; release
  LIN {X -15850.033,Y -1181.101,Z 62.331,A 131.29142,B 0.00000,C 180.00000} ; retreat
  ; Step 1044, bar 3042
  LIN {X -15450.033,Y -1181.101,Z 967.962,A 131.29142,B 0.00000,C 180.00000} ; outside
  LIN {X -15450.033,Y -1181.101,Z 12.331,A 131.29142,B 0.00000,C 180.00000} ; preinsert
  LIN {X -15450.033,Y -1181.101,Z -237.669,A 131.29142,B 0.00000,C 180.00000} ; insert
  LIN {X -15450.033,Y -1181.101,Z -237.669,A 131.29142,B 0.00000,C 180.00000} ; release
  LIN {X -15450.033,Y -1181.101,Z 62.331,A 131.29142,B 0.00000,C 180.00000} ; retreat
  ; Step 1045, bar 3058
  LIN {X 15450.033,Y 1181.101,Z 967.962,A -48.70858,B 0.00000,C 180.00000} ; outside
  LIN {X 15450.033,Y 1181.101,Z 12.331,A -48.70858,B 0.00000,C 180.00000} ; preinsert
  LIN {X 15450.033,Y 1181.101,Z -237.669,A -48.70858,B 0.00000,C 180.00000} ; insert
  LIN {X 15450.033,Y 1181.101,Z -237.669,A -48.70858,B 0.00000,C 180.00000} ; release
  LIN {X 15450.033,Y 1181.101,Z 62.331,A -48.70858,B 0.00000,C 180.00000} ; retreat
  ; Step 1046, bar 3064
  LIN {X 15850.033,Y 1181.101,Z 967.962,A -48.70858,B 0.00000,C 180.00000} ; outside
  LIN {X 15850.033,Y 1181.101,Z 12.331,A -48.70858,B 0.00000,C 180.00000} ; preinsert
  LIN {X 15850.033,Y 1181.101,Z -237.669,A -48.70858,B 0.00000,C 180.00000} ; insert
  LIN {X 15850.033,Y 1181.101,Z -237.669,A -48.70858,B 0.00000,C 180.00000} ; release
  LIN {X 15850.033,Y 1181.101,Z 62.331,A -48.70858,B 0.00000,C 180.00000} ; retreat
  ; Step 1047, bar 3070
  LIN {X 16250.033,Y 1181.101,Z 967.962,A -48.70858,B 0.00000,C 180.00000} ; outside
  LIN {X 16250.033,Y 1181.101,Z 12.331,A -48.70858,B 0.00000,C 180.00000} ; preinsert
  LIN {X 16250.033,Y 1181.101,Z -237.669,A -48.70858,B 0.00000,C 180.00000} ; insert
  LIN {X 16250.033,Y 1181.101,Z -237.669,A -48.70858,B 0.00000,C 180.00000} ; release
  LIN {X 16250.033,Y 1181.101,Z 62.331,A -48.70858,B 0.00000,C 180.00000} ; retreat
  ; Step 1048, bar 887
  LIN {X 15549.900,Y -1914.437,Z 1107.719,A 90.00016,B 0.00000,C 180.00000} ; outside
  LIN {X 15549.900,Y -1914.437,Z 173.363,A 90.00016,B 0.00000,C 180.00000} ; preinsert
  LIN {X 15549.900,Y -1914.437,Z -76.637,A 90.00016,B 0.00000,C 180.00000} ; insert
  LIN {X 15549.900,Y -1914.437,Z -76.637,A 90.00016,B 0.00000,C 180.00000} ; release
  LIN {X 15549.900,Y -1914.437,Z 223.363,A 90.00016,B 0.00000,C 180.00000} ; retreat
  ; Step 1049, bar 891
  LIN {X -15549.900,Y -1914.437,Z 1107.719,A 89.99984,B 0.00000,C 180.00000} ; outside
  LIN {X -15549.900,Y -1914.437,Z 173.363,A 89.99984,B 0.00000,C 180.00000} ; preinsert
  LIN {X -15549.900,Y -1914.437,Z -76.637,A 89.99984,B 0.00000,C 180.00000} ; insert
  LIN {X -15549.900,Y -1914.437,Z -76.637,A 89.99984,B 0.00000,C 180.00000} ; release
  LIN {X -15549.900,Y -1914.437,Z 223.363,A 89.99984,B 0.00000,C 180.00000} ; retreat
  ; Step 1050, bar 886
  LIN {X 14549.900,Y -1914.437,Z 1107.719,A 90.00016,B 0.00000,C 180.00000} ; outside
  LIN {X 14549.900,Y -1914.437,Z 173.363,A 90.00016,B 0.00000,C 180.00000} ; preinsert
  LIN {X 14549.900,Y -1914.437,Z -76.637,A 90.00016,B 0.00000,C 180.00000} ; insert
  LIN {X 14549.900,Y -1914.437,Z -76.637,A 90.00016,B 0.00000,C 180.00000} ; release
  LIN {X 14549.900,Y -1914.437,Z 223.363,A 90.00016,B 0.00000,C 180.00000} ; retreat
  ; Step 1051, bar 890
  LIN {X -14549.900,Y -1914.437,Z 1107.719,A 89.99984,B 0.00000,C 180.00000} ; outside
  LIN {X -14549.900,Y -1914.437,Z 173.363,A 89.99984,B 0.00000,C 180.00000} ; preinsert
  LIN {X -14549.900,Y -1914.437,Z -76.637,A 89.99984,B 0.00000,C 180.00000} ; insert
  LIN {X -14549.900,Y -1914.437,Z -76.637,A 89.99984,B 0.00000,C 180.00000} ; release
  LIN {X -14549.900,Y -1914.437,Z 223.363,A 89.99984,B 0.00000,C 180.00000} ; retreat
  ; Step 1052, bar 889
  LIN {X -15549.900,Y 1914.437,Z 1107.719,A -89.99984,B 0.00000,C 180.00000} ; outside
  LIN {X -15549.900,Y 1914.437,Z 173.363,A -89.99984,B 0.00000,C 180.00000} ; preinsert
  LIN {X -15549.900,Y 1914.437,Z -76.637,A -89.99984,B 0.00000,C 180.00000} ; insert
  LIN {X -15549.900,Y 1914.437,Z -76.637,A -89.99984,B 0.00000,C 180.00000} ; release
  LIN {X -15549.900,Y 1914.437,Z 223.363,A -89.99984,B 0.00000,C 180.00000} ; retreat
  ; Step 1053, bar 885
  LIN {X 15549.900,Y 1914.437,Z 1107.719,A -90.00016,B 0.00000,C -180.00000} ; outside
  LIN {X 15549.900,Y 1914.437,Z 173.363,A -90.00016,B 0.00000,C -180.00000} ; preinsert
  LIN {X 15549.900,Y 1914.437,Z -76.637,A -90.00016,B 0.00000,C -180.00000} ; insert
  LIN {X 15549.900,Y 1914.437,Z -76.637,A -90.00016,B 0.00000,C -180.00000} ; release
  LIN {X 15549.900,Y 1914.437,Z 223.363,A -90.00016,B 0.00000,C -180.00000} ; retreat
  ; Step 1054, bar 888
  LIN {X -14549.900,Y 1914.437,Z 1107.719,A -89.99984,B 0.00000,C 180.00000} ; outside
  LIN {X -14549.900,Y 1914.437,Z 173.363,A -89.99984,B 0.00000,C 180.00000} ; preinsert
  LIN {X -14549.900,Y 1914.437,Z -76.637,A -89.99984,B 0.00000,C 180.00000} ; insert
  LIN {X -14549.900,Y 1914.437,Z -76.637,A -89.99984,B 0.00000,C 180.00000} ; release
  LIN {X -14549.900,Y 1914.437,Z 223.363,A -89.99984,B 0.00000,C 180.00000} ; retreat
  ; Step 1055, bar 884
  LIN {X 14549.900,Y 1914.437,Z 1107.719,A -90.00016,B 0.00000,C -180.00000} ; outside
  LIN {X 14549.900,Y 1914.437,Z 173.363,A -90.00016,B 0.00000,C -180.00000} ; preinsert
  LIN {X 14549.900,Y 1914.437,Z -76.637,A -90.00016,B 0.00000,C -180.00000} ; insert
  LIN {X 14549.900,Y 1914.437,Z -76.637,A -90.00016,B 0.00000,C -180.00000} ; release
  LIN {X 14549.900,Y 1914.437,Z 223.363,A -90.00016,B 0.00000,C -180.00000} ; retreat
  ; Step 1056, bar 302
  LIN {X 0.000,Y -3265.000,Z 1124.718,A 0.00000,B 0.00000,C 180.00000} ; outside
  LIN {X 0.000,Y -3265.000,Z 186.669,A 0.00000,B 0.00000,C 180.00000} ; preinsert
  LIN {X 0.000,Y -3265.000,Z -63.331,A 0.00000,B 0.00000,C 180.00000} ; insert
  LIN {X 0.000,Y -3265.000,Z -63.331,A 0.00000,B 0.00000,C 180.00000} ; release
  LIN {X 0.000,Y -3265.000,Z 236.669,A 0.00000,B 0.00000,C 180.00000} ; retreat
  ; Step 1057, bar 329
  LIN {X 0.000,Y 3265.000,Z 1124.718,A 0.00000,B 0.00000,C 180.00000} ; outside
  LIN {X 0.000,Y 3265.000,Z 186.669,A 0.00000,B 0.00000,C 180.00000} ; preinsert
  LIN {X 0.000,Y 3265.000,Z -63.331,A 0.00000,B 0.00000,C 180.00000} ; insert
  LIN {X 0.000,Y 3265.000,Z -63.331,A 0.00000,B 0.00000,C 180.00000} ; release
  LIN {X 0.000,Y 3265.000,Z 236.669,A 0.00000,B 0.00000,C 180.00000} ; retreat
  ; Step 1058, bar 303
  LIN {X 0.000,Y -3355.000,Z 1125.716,A 0.00000,B 0.00000,C 180.00000} ; outside
  LIN {X 0.000,Y -3355.000,Z 187.168,A 0.00000,B 0.00000,C 180.00000} ; preinsert
  LIN {X 0.000,Y -3355.000,Z -62.832,A 0.00000,B 0.00000,C 180.00000} ; insert
  LIN {X 0.000,Y -3355.000,Z -62.832,A 0.00000,B 0.00000,C 180.00000} ; release
  LIN {X 0.000,Y -3355.000,Z 237.168,A 0.00000,B 0.00000,C 180.00000} ; retreat
  ; Step 1059, bar 330
  LIN {X 0.000,Y 3355.000,Z 1125.716,A 0.00000,B 0.00000,C 180.00000} ; outside
  LIN {X 0.000,Y 3355.000,Z 187.168,A 0.00000,B 0.00000,C 180.00000} ; preinsert
  LIN {X 0.000,Y 3355.000,Z -62.832,A 0.00000,B 0.00000,C 180.00000} ; insert
  LIN {X 0.000,Y 3355.000,Z -62.832,A 0.00000,B 0.00000,C 180.00000} ; release
  LIN {X 0.000,Y 3355.000,Z 237.168,A 0.00000,B 0.00000,C 180.00000} ; retreat
  ; Step 1060, bar 3103
  LIN {X -15204.133,Y -141.217,Z 1079.276,A -179.87076,B 0.00000,C -180.00000} ; outside
  LIN {X -15204.133,Y -141.217,Z 113.892,A -179.87076,B 0.00000,C -180.00000} ; preinsert
  LIN {X -15204.133,Y -141.217,Z -136.108,A -179.87076,B 0.00000,C -180.00000} ; insert
  LIN {X -15204.133,Y -141.217,Z -136.108,A -179.87076,B 0.00000,C -180.00000} ; release
  LIN {X -15204.133,Y -141.217,Z 163.892,A -179.87076,B 0.00000,C -180.00000} ; retreat
  ; Step 1061, bar 3093
  LIN {X 15204.133,Y -141.217,Z 1079.276,A -0.12924,B 0.00000,C 180.00000} ; outside
  LIN {X 15204.133,Y -141.217,Z 113.892,A -0.12924,B 0.00000,C 180.00000} ; preinsert
  LIN {X 15204.133,Y -141.217,Z -136.108,A -0.12924,B 0.00000,C 180.00000} ; insert
  LIN {X 15204.133,Y -141.217,Z -136.108,A -0.12924,B 0.00000,C 180.00000} ; release
  LIN {X 15204.133,Y -141.217,Z 163.892,A -0.12924,B 0.00000,C 180.00000} ; retreat
  ; Step 1062, bar 3098
  LIN {X -15204.133,Y 141.217,Z 1079.276,A 179.87076,B 0.00000,C -180.00000} ; outside
  LIN {X -15204.133,Y 141.217,Z 113.892,A 179.87076,B 0.00000,C -180.00000} ; preinsert
  LIN {X -15204.133,Y 141.217,Z -136.108,A 179.87076,B 0.00000,C -180.00000} ; insert
  LIN {X -15204.133,Y 141.217,Z -136.108,A 179.87076,B 0.00000,C -180.00000} ; release
  LIN {X -15204.133,Y 141.217,Z 163.892,A 179.87076,B 0.00000,C -180.00000} ; retreat
  ; Step 1063, bar 3088
  LIN {X 15204.133,Y 141.217,Z 1079.276,A 0.12924,B 0.00000,C 180.00000} ; outside
  LIN {X 15204.133,Y 141.217,Z 113.892,A 0.12924,B 0.00000,C 180.00000} ; preinsert
  LIN {X 15204.133,Y 141.217,Z -136.108,A 0.12924,B 0.00000,C 180.00000} ; insert
  LIN {X 15204.133,Y 141.217,Z -136.108,A 0.12924,B 0.00000,C 180.00000} ; release
  LIN {X 15204.133,Y 141.217,Z 163.892,A 0.12924,B 0.00000,C 180.00000} ; retreat
  ; Step 1064, bar 2753
  LIN {X -1124.942,Y -1181.101,Z 999.474,A 91.55051,B 0.00000,C 180.00000} ; outside
  LIN {X -1124.942,Y -1181.101,Z 60.229,A 91.55051,B 0.00000,C 180.00000} ; preinsert
  LIN {X -1124.942,Y -1181.101,Z -189.771,A 91.55051,B 0.00000,C 180.00000} ; insert
  LIN {X -1124.942,Y -1181.101,Z -189.771,A 91.55051,B 0.00000,C 180.00000} ; release
  LIN {X -1124.942,Y -1181.101,Z 110.229,A 91.55051,B 0.00000,C 180.00000} ; retreat
  ; Step 1065, bar 2750
  LIN {X -374.942,Y -1181.101,Z 999.474,A 91.55051,B 0.00000,C -180.00000} ; outside
  LIN {X -374.942,Y -1181.101,Z 60.229,A 91.55051,B 0.00000,C -180.00000} ; preinsert
  LIN {X -374.942,Y -1181.101,Z -189.771,A 91.55051,B 0.00000,C -180.00000} ; insert
  LIN {X -374.942,Y -1181.101,Z -189.771,A 91.55051,B 0.00000,C -180.00000} ; release
  LIN {X -374.942,Y -1181.101,Z 110.229,A 91.55051,B 0.00000,C -180.00000} ; retreat
  ; Step 1066, bar 2756
  LIN {X -1874.942,Y -1181.101,Z 999.474,A 91.55051,B 0.00000,C 180.00000} ; outside
  LIN {X -1874.942,Y -1181.101,Z 60.229,A 91.55051,B 0.00000,C 180.00000} ; preinsert
  LIN {X -1874.942,Y -1181.101,Z -189.771,A 91.55051,B 0.00000,C 180.00000} ; insert
  LIN {X -1874.942,Y -1181.101,Z -189.771,A 91.55051,B 0.00000,C 180.00000} ; release
  LIN {X -1874.942,Y -1181.101,Z 110.229,A 91.55051,B 0.00000,C 180.00000} ; retreat
  ; Step 1067, bar 2759
  LIN {X -2624.942,Y -1181.101,Z 999.474,A 91.55051,B 0.00000,C 180.00000} ; outside
  LIN {X -2624.942,Y -1181.101,Z 60.229,A 91.55051,B 0.00000,C 180.00000} ; preinsert
  LIN {X -2624.942,Y -1181.101,Z -189.771,A 91.55051,B 0.00000,C 180.00000} ; insert
  LIN {X -2624.942,Y -1181.101,Z -189.771,A 91.55051,B 0.00000,C 180.00000} ; release
  LIN {X -2624.942,Y -1181.101,Z 110.229,A 91.55051,B 0.00000,C 180.00000} ; retreat
  ; Step 1068, bar 2762
  LIN {X -3374.942,Y -1181.101,Z 999.474,A 91.55051,B 0.00000,C 180.00000} ; outside
  LIN {X -3374.942,Y -1181.101,Z 60.229,A 91.55051,B 0.00000,C 180.00000} ; preinsert
  LIN {X -3374.942,Y -1181.101,Z -189.771,A 91.55051,B 0.00000,C 180.00000} ; insert
  LIN {X -3374.942,Y -1181.101,Z -189.771,A 91.55051,B 0.00000,C 180.00000} ; release
  LIN {X -3374.942,Y -1181.101,Z 110.229,A 91.55051,B 0.00000,C 180.00000} ; retreat
  ; Step 1069, bar 2765
  LIN {X -4124.942,Y -1181.101,Z 999.474,A 91.55051,B 0.00000,C 180.00000} ; outside
  LIN {X -4124.942,Y -1181.101,Z 60.229,A 91.55051,B 0.00000,C 180.00000} ; preinsert
  LIN {X -4124.942,Y -1181.101,Z -189.771,A 91.55051,B 0.00000,C 180.00000} ; insert
  LIN {X -4124.942,Y -1181.101,Z -189.771,A 91.55051,B 0.00000,C 180.00000} ; release
  LIN {X -4124.942,Y -1181.101,Z 110.229,A 91.55051,B 0.00000,C 180.00000} ; retreat
  ; Step 1070, bar 2768
  LIN {X -4874.942,Y -1181.101,Z 999.474,A 91.55051,B 0.00000,C 180.00000} ; outside
  LIN {X -4874.942,Y -1181.101,Z 60.229,A 91.55051,B 0.00000,C 180.00000} ; preinsert
  LIN {X -4874.942,Y -1181.101,Z -189.771,A 91.55051,B 0.00000,C 180.00000} ; insert
  LIN {X -4874.942,Y -1181.101,Z -189.771,A 91.55051,B 0.00000,C 180.00000} ; release
  LIN {X -4874.942,Y -1181.101,Z 110.229,A 91.55051,B 0.00000,C 180.00000} ; retreat
  ; Step 1071, bar 2771
  LIN {X -5624.942,Y -1181.101,Z 999.474,A 91.55051,B 0.00000,C 180.00000} ; outside
  LIN {X -5624.942,Y -1181.101,Z 60.229,A 91.55051,B 0.00000,C 180.00000} ; preinsert
  LIN {X -5624.942,Y -1181.101,Z -189.771,A 91.55051,B 0.00000,C 180.00000} ; insert
  LIN {X -5624.942,Y -1181.101,Z -189.771,A 91.55051,B 0.00000,C 180.00000} ; release
  LIN {X -5624.942,Y -1181.101,Z 110.229,A 91.55051,B 0.00000,C 180.00000} ; retreat
  ; Step 1072, bar 2774
  LIN {X -6374.942,Y -1181.101,Z 999.474,A 91.55051,B 0.00000,C 180.00000} ; outside
  LIN {X -6374.942,Y -1181.101,Z 60.229,A 91.55051,B 0.00000,C 180.00000} ; preinsert
  LIN {X -6374.942,Y -1181.101,Z -189.771,A 91.55051,B 0.00000,C 180.00000} ; insert
  LIN {X -6374.942,Y -1181.101,Z -189.771,A 91.55051,B 0.00000,C 180.00000} ; release
  LIN {X -6374.942,Y -1181.101,Z 110.229,A 91.55051,B 0.00000,C 180.00000} ; retreat
  ; Step 1073, bar 2777
  LIN {X -7124.942,Y -1181.101,Z 999.474,A 91.55051,B 0.00000,C 180.00000} ; outside
  LIN {X -7124.942,Y -1181.101,Z 60.229,A 91.55051,B 0.00000,C 180.00000} ; preinsert
  LIN {X -7124.942,Y -1181.101,Z -189.771,A 91.55051,B 0.00000,C 180.00000} ; insert
  LIN {X -7124.942,Y -1181.101,Z -189.771,A 91.55051,B 0.00000,C 180.00000} ; release
  LIN {X -7124.942,Y -1181.101,Z 110.229,A 91.55051,B 0.00000,C 180.00000} ; retreat
  ; Step 1074, bar 2780
  LIN {X -7874.942,Y -1181.101,Z 999.474,A 91.55051,B 0.00000,C 180.00000} ; outside
  LIN {X -7874.942,Y -1181.101,Z 60.229,A 91.55051,B 0.00000,C 180.00000} ; preinsert
  LIN {X -7874.942,Y -1181.101,Z -189.771,A 91.55051,B 0.00000,C 180.00000} ; insert
  LIN {X -7874.942,Y -1181.101,Z -189.771,A 91.55051,B 0.00000,C 180.00000} ; release
  LIN {X -7874.942,Y -1181.101,Z 110.229,A 91.55051,B 0.00000,C 180.00000} ; retreat
  ; Step 1075, bar 2783
  LIN {X -8624.942,Y -1181.101,Z 999.474,A 91.55051,B 0.00000,C 180.00000} ; outside
  LIN {X -8624.942,Y -1181.101,Z 60.229,A 91.55051,B 0.00000,C 180.00000} ; preinsert
  LIN {X -8624.942,Y -1181.101,Z -189.771,A 91.55051,B 0.00000,C 180.00000} ; insert
  LIN {X -8624.942,Y -1181.101,Z -189.771,A 91.55051,B 0.00000,C 180.00000} ; release
  LIN {X -8624.942,Y -1181.101,Z 110.229,A 91.55051,B 0.00000,C 180.00000} ; retreat
  ; Step 1076, bar 2786
  LIN {X -9374.942,Y -1181.101,Z 999.474,A 91.55051,B 0.00000,C 180.00000} ; outside
  LIN {X -9374.942,Y -1181.101,Z 60.229,A 91.55051,B 0.00000,C 180.00000} ; preinsert
  LIN {X -9374.942,Y -1181.101,Z -189.771,A 91.55051,B 0.00000,C 180.00000} ; insert
  LIN {X -9374.942,Y -1181.101,Z -189.771,A 91.55051,B 0.00000,C 180.00000} ; release
  LIN {X -9374.942,Y -1181.101,Z 110.229,A 91.55051,B 0.00000,C 180.00000} ; retreat
  ; Step 1077, bar 2789
  LIN {X -10124.942,Y -1181.101,Z 999.474,A 91.55051,B 0.00000,C 180.00000} ; outside
  LIN {X -10124.942,Y -1181.101,Z 60.229,A 91.55051,B 0.00000,C 180.00000} ; preinsert
  LIN {X -10124.942,Y -1181.101,Z -189.771,A 91.55051,B 0.00000,C 180.00000} ; insert
  LIN {X -10124.942,Y -1181.101,Z -189.771,A 91.55051,B 0.00000,C 180.00000} ; release
  LIN {X -10124.942,Y -1181.101,Z 110.229,A 91.55051,B 0.00000,C 180.00000} ; retreat
  ; Step 1078, bar 2792
  LIN {X -10874.942,Y -1181.101,Z 999.474,A 91.55051,B 0.00000,C 180.00000} ; outside
  LIN {X -10874.942,Y -1181.101,Z 60.229,A 91.55051,B 0.00000,C 180.00000} ; preinsert
  LIN {X -10874.942,Y -1181.101,Z -189.771,A 91.55051,B 0.00000,C 180.00000} ; insert
  LIN {X -10874.942,Y -1181.101,Z -189.771,A 91.55051,B 0.00000,C 180.00000} ; release
  LIN {X -10874.942,Y -1181.101,Z 110.229,A 91.55051,B 0.00000,C 180.00000} ; retreat
  ; Step 1079, bar 2795
  LIN {X -11624.942,Y -1181.101,Z 999.474,A 91.55051,B 0.00000,C 180.00000} ; outside
  LIN {X -11624.942,Y -1181.101,Z 60.229,A 91.55051,B 0.00000,C 180.00000} ; preinsert
  LIN {X -11624.942,Y -1181.101,Z -189.771,A 91.55051,B 0.00000,C 180.00000} ; insert
  LIN {X -11624.942,Y -1181.101,Z -189.771,A 91.55051,B 0.00000,C 180.00000} ; release
  LIN {X -11624.942,Y -1181.101,Z 110.229,A 91.55051,B 0.00000,C 180.00000} ; retreat
  ; Step 1080, bar 2637
  LIN {X 374.942,Y 1181.101,Z 999.474,A -88.44949,B 0.00000,C 180.00000} ; outside
  LIN {X 374.942,Y 1181.101,Z 60.229,A -88.44949,B 0.00000,C 180.00000} ; preinsert
  LIN {X 374.942,Y 1181.101,Z -189.771,A -88.44949,B 0.00000,C 180.00000} ; insert
  LIN {X 374.942,Y 1181.101,Z -189.771,A -88.44949,B 0.00000,C 180.00000} ; release
  LIN {X 374.942,Y 1181.101,Z 110.229,A -88.44949,B 0.00000,C 180.00000} ; retreat
  ; Step 1081, bar 2639
  LIN {X 1124.942,Y 1181.101,Z 999.474,A -88.44949,B 0.00000,C -180.00000} ; outside
  LIN {X 1124.942,Y 1181.101,Z 60.229,A -88.44949,B 0.00000,C -180.00000} ; preinsert
  LIN {X 1124.942,Y 1181.101,Z -189.771,A -88.44949,B 0.00000,C -180.00000} ; insert
  LIN {X 1124.942,Y 1181.101,Z -189.771,A -88.44949,B 0.00000,C -180.00000} ; release
  LIN {X 1124.942,Y 1181.101,Z 110.229,A -88.44949,B 0.00000,C -180.00000} ; retreat
  ; Step 1082, bar 2642
  LIN {X 1874.942,Y 1181.101,Z 999.474,A -88.44949,B 0.00000,C -180.00000} ; outside
  LIN {X 1874.942,Y 1181.101,Z 60.229,A -88.44949,B 0.00000,C -180.00000} ; preinsert
  LIN {X 1874.942,Y 1181.101,Z -189.771,A -88.44949,B 0.00000,C -180.00000} ; insert
  LIN {X 1874.942,Y 1181.101,Z -189.771,A -88.44949,B 0.00000,C -180.00000} ; release
  LIN {X 1874.942,Y 1181.101,Z 110.229,A -88.44949,B 0.00000,C -180.00000} ; retreat
  ; Step 1083, bar 2645
  LIN {X 2624.942,Y 1181.101,Z 999.474,A -88.44949,B 0.00000,C 180.00000} ; outside
  LIN {X 2624.942,Y 1181.101,Z 60.229,A -88.44949,B 0.00000,C 180.00000} ; preinsert
  LIN {X 2624.942,Y 1181.101,Z -189.771,A -88.44949,B 0.00000,C 180.00000} ; insert
  LIN {X 2624.942,Y 1181.101,Z -189.771,A -88.44949,B 0.00000,C 180.00000} ; release
  LIN {X 2624.942,Y 1181.101,Z 110.229,A -88.44949,B 0.00000,C 180.00000} ; retreat
  ; Step 1084, bar 2648
  LIN {X 3374.942,Y 1181.101,Z 999.474,A -88.44949,B 0.00000,C 180.00000} ; outside
  LIN {X 3374.942,Y 1181.101,Z 60.229,A -88.44949,B 0.00000,C 180.00000} ; preinsert
  LIN {X 3374.942,Y 1181.101,Z -189.771,A -88.44949,B 0.00000,C 180.00000} ; insert
  LIN {X 3374.942,Y 1181.101,Z -189.771,A -88.44949,B 0.00000,C 180.00000} ; release
  LIN {X 3374.942,Y 1181.101,Z 110.229,A -88.44949,B 0.00000,C 180.00000} ; retreat
  ; Step 1085, bar 2651
  LIN {X 4124.942,Y 1181.101,Z 999.474,A -88.44949,B 0.00000,C 180.00000} ; outside
  LIN {X 4124.942,Y 1181.101,Z 60.229,A -88.44949,B 0.00000,C 180.00000} ; preinsert
  LIN {X 4124.942,Y 1181.101,Z -189.771,A -88.44949,B 0.00000,C 180.00000} ; insert
  LIN {X 4124.942,Y 1181.101,Z -189.771,A -88.44949,B 0.00000,C 180.00000} ; release
  LIN {X 4124.942,Y 1181.101,Z 110.229,A -88.44949,B 0.00000,C 180.00000} ; retreat
  ; Step 1086, bar 2654
  LIN {X 4874.942,Y 1181.101,Z 999.474,A -88.44949,B 0.00000,C 180.00000} ; outside
  LIN {X 4874.942,Y 1181.101,Z 60.229,A -88.44949,B 0.00000,C 180.00000} ; preinsert
  LIN {X 4874.942,Y 1181.101,Z -189.771,A -88.44949,B 0.00000,C 180.00000} ; insert
  LIN {X 4874.942,Y 1181.101,Z -189.771,A -88.44949,B 0.00000,C 180.00000} ; release
  LIN {X 4874.942,Y 1181.101,Z 110.229,A -88.44949,B 0.00000,C 180.00000} ; retreat
  ; Step 1087, bar 2657
  LIN {X 5624.942,Y 1181.101,Z 999.474,A -88.44949,B 0.00000,C 180.00000} ; outside
  LIN {X 5624.942,Y 1181.101,Z 60.229,A -88.44949,B 0.00000,C 180.00000} ; preinsert
  LIN {X 5624.942,Y 1181.101,Z -189.771,A -88.44949,B 0.00000,C 180.00000} ; insert
  LIN {X 5624.942,Y 1181.101,Z -189.771,A -88.44949,B 0.00000,C 180.00000} ; release
  LIN {X 5624.942,Y 1181.101,Z 110.229,A -88.44949,B 0.00000,C 180.00000} ; retreat
  ; Step 1088, bar 2660
  LIN {X 6374.942,Y 1181.101,Z 999.474,A -88.44949,B 0.00000,C 180.00000} ; outside
  LIN {X 6374.942,Y 1181.101,Z 60.229,A -88.44949,B 0.00000,C 180.00000} ; preinsert
  LIN {X 6374.942,Y 1181.101,Z -189.771,A -88.44949,B 0.00000,C 180.00000} ; insert
  LIN {X 6374.942,Y 1181.101,Z -189.771,A -88.44949,B 0.00000,C 180.00000} ; release
  LIN {X 6374.942,Y 1181.101,Z 110.229,A -88.44949,B 0.00000,C 180.00000} ; retreat
  ; Step 1089, bar 2663
  LIN {X 7124.942,Y 1181.101,Z 999.474,A -88.44949,B 0.00000,C 180.00000} ; outside
  LIN {X 7124.942,Y 1181.101,Z 60.229,A -88.44949,B 0.00000,C 180.00000} ; preinsert
  LIN {X 7124.942,Y 1181.101,Z -189.771,A -88.44949,B 0.00000,C 180.00000} ; insert
  LIN {X 7124.942,Y 1181.101,Z -189.771,A -88.44949,B 0.00000,C 180.00000} ; release
  LIN {X 7124.942,Y 1181.101,Z 110.229,A -88.44949,B 0.00000,C 180.00000} ; retreat
  ; Step 1090, bar 2666
  LIN {X 7874.942,Y 1181.101,Z 999.474,A -88.44949,B 0.00000,C 180.00000} ; outside
  LIN {X 7874.942,Y 1181.101,Z 60.229,A -88.44949,B 0.00000,C 180.00000} ; preinsert
  LIN {X 7874.942,Y 1181.101,Z -189.771,A -88.44949,B 0.00000,C 180.00000} ; insert
  LIN {X 7874.942,Y 1181.101,Z -189.771,A -88.44949,B 0.00000,C 180.00000} ; release
  LIN {X 7874.942,Y 1181.101,Z 110.229,A -88.44949,B 0.00000,C 180.00000} ; retreat
  ; Step 1091, bar 2669
  LIN {X 8624.942,Y 1181.101,Z 999.474,A -88.44949,B 0.00000,C 180.00000} ; outside
  LIN {X 8624.942,Y 1181.101,Z 60.229,A -88.44949,B 0.00000,C 180.00000} ; preinsert
  LIN {X 8624.942,Y 1181.101,Z -189.771,A -88.44949,B 0.00000,C 180.00000} ; insert
  LIN {X 8624.942,Y 1181.101,Z -189.771,A -88.44949,B 0.00000,C 180.00000} ; release
  LIN {X 8624.942,Y 1181.101,Z 110.229,A -88.44949,B 0.00000,C 180.00000} ; retreat
  ; Step 1092, bar 2672
  LIN {X 9374.942,Y 1181.101,Z 999.474,A -88.44949,B 0.00000,C 180.00000} ; outside
  LIN {X 9374.942,Y 1181.101,Z 60.229,A -88.44949,B 0.00000,C 180.00000} ; preinsert
  LIN {X 9374.942,Y 1181.101,Z -189.771,A -88.44949,B 0.00000,C 180.00000} ; insert
  LIN {X 9374.942,Y 1181.101,Z -189.771,A -88.44949,B 0.00000,C 180.00000} ; release
  LIN {X 9374.942,Y 1181.101,Z 110.229,A -88.44949,B 0.00000,C 180.00000} ; retreat
  ; Step 1093, bar 2675
  LIN {X 10124.942,Y 1181.101,Z 999.474,A -88.44949,B 0.00000,C 180.00000} ; outside
  LIN {X 10124.942,Y 1181.101,Z 60.229,A -88.44949,B 0.00000,C 180.00000} ; preinsert
  LIN {X 10124.942,Y 1181.101,Z -189.771,A -88.44949,B 0.00000,C 180.00000} ; insert
  LIN {X 10124.942,Y 1181.101,Z -189.771,A -88.44949,B 0.00000,C 180.00000} ; release
  LIN {X 10124.942,Y 1181.101,Z 110.229,A -88.44949,B 0.00000,C 180.00000} ; retreat
  ; Step 1094, bar 2678
  LIN {X 10874.942,Y 1181.101,Z 999.474,A -88.44949,B 0.00000,C 180.00000} ; outside
  LIN {X 10874.942,Y 1181.101,Z 60.229,A -88.44949,B 0.00000,C 180.00000} ; preinsert
  LIN {X 10874.942,Y 1181.101,Z -189.771,A -88.44949,B 0.00000,C 180.00000} ; insert
  LIN {X 10874.942,Y 1181.101,Z -189.771,A -88.44949,B 0.00000,C 180.00000} ; release
  LIN {X 10874.942,Y 1181.101,Z 110.229,A -88.44949,B 0.00000,C 180.00000} ; retreat
  ; Step 1095, bar 2681
  LIN {X 11624.942,Y 1181.101,Z 999.474,A -88.44949,B 0.00000,C 180.00000} ; outside
  LIN {X 11624.942,Y 1181.101,Z 60.229,A -88.44949,B 0.00000,C 180.00000} ; preinsert
  LIN {X 11624.942,Y 1181.101,Z -189.771,A -88.44949,B 0.00000,C 180.00000} ; insert
  LIN {X 11624.942,Y 1181.101,Z -189.771,A -88.44949,B 0.00000,C 180.00000} ; release
  LIN {X 11624.942,Y 1181.101,Z 110.229,A -88.44949,B 0.00000,C 180.00000} ; retreat
  ; Step 1096, bar 2799
  LIN {X 374.942,Y -1181.101,Z 999.474,A 88.44949,B 0.00000,C 180.00000} ; outside
  LIN {X 374.942,Y -1181.101,Z 60.229,A 88.44949,B 0.00000,C 180.00000} ; preinsert
  LIN {X 374.942,Y -1181.101,Z -189.771,A 88.44949,B 0.00000,C 180.00000} ; insert
  LIN {X 374.942,Y -1181.101,Z -189.771,A 88.44949,B 0.00000,C 180.00000} ; release
  LIN {X 374.942,Y -1181.101,Z 110.229,A 88.44949,B 0.00000,C 180.00000} ; retreat
  ; Step 1097, bar 2801
  LIN {X 1124.942,Y -1181.101,Z 999.474,A 88.44949,B 0.00000,C -180.00000} ; outside
  LIN {X 1124.942,Y -1181.101,Z 60.229,A 88.44949,B 0.00000,C -180.00000} ; preinsert
  LIN {X 1124.942,Y -1181.101,Z -189.771,A 88.44949,B 0.00000,C -180.00000} ; insert
  LIN {X 1124.942,Y -1181.101,Z -189.771,A 88.44949,B 0.00000,C -180.00000} ; release
  LIN {X 1124.942,Y -1181.101,Z 110.229,A 88.44949,B 0.00000,C -180.00000} ; retreat
  ; Step 1098, bar 2804
  LIN {X 1874.942,Y -1181.101,Z 999.474,A 88.44949,B 0.00000,C -180.00000} ; outside
  LIN {X 1874.942,Y -1181.101,Z 60.229,A 88.44949,B 0.00000,C -180.00000} ; preinsert
  LIN {X 1874.942,Y -1181.101,Z -189.771,A 88.44949,B 0.00000,C -180.00000} ; insert
  LIN {X 1874.942,Y -1181.101,Z -189.771,A 88.44949,B 0.00000,C -180.00000} ; release
  LIN {X 1874.942,Y -1181.101,Z 110.229,A 88.44949,B 0.00000,C -180.00000} ; retreat
  ; Step 1099, bar 2807
  LIN {X 2624.942,Y -1181.101,Z 999.474,A 88.44949,B 0.00000,C 180.00000} ; outside
  LIN {X 2624.942,Y -1181.101,Z 60.229,A 88.44949,B 0.00000,C 180.00000} ; preinsert
  LIN {X 2624.942,Y -1181.101,Z -189.771,A 88.44949,B 0.00000,C 180.00000} ; insert
  LIN {X 2624.942,Y -1181.101,Z -189.771,A 88.44949,B 0.00000,C 180.00000} ; release
  LIN {X 2624.942,Y -1181.101,Z 110.229,A 88.44949,B 0.00000,C 180.00000} ; retreat
  ; Step 1100, bar 2810
  LIN {X 3374.942,Y -1181.101,Z 999.474,A 88.44949,B 0.00000,C 180.00000} ; outside
  LIN {X 3374.942,Y -1181.101,Z 60.229,A 88.44949,B 0.00000,C 180.00000} ; preinsert
  LIN {X 3374.942,Y -1181.101,Z -189.771,A 88.44949,B 0.00000,C 180.00000} ; insert
  LIN {X 3374.942,Y -1181.101,Z -189.771,A 88.44949,B 0.00000,C 180.00000} ; release
  LIN {X 3374.942,Y -1181.101,Z 110.229,A 88.44949,B 0.00000,C 180.00000} ; retreat
  ; Step 1101, bar 2813
  LIN {X 4124.942,Y -1181.101,Z 999.474,A 88.44949,B 0.00000,C 180.00000} ; outside
  LIN {X 4124.942,Y -1181.101,Z 60.229,A 88.44949,B 0.00000,C 180.00000} ; preinsert
  LIN {X 4124.942,Y -1181.101,Z -189.771,A 88.44949,B 0.00000,C 180.00000} ; insert
  LIN {X 4124.942,Y -1181.101,Z -189.771,A 88.44949,B 0.00000,C 180.00000} ; release
  LIN {X 4124.942,Y -1181.101,Z 110.229,A 88.44949,B 0.00000,C 180.00000} ; retreat
  ; Step 1102, bar 2816
  LIN {X 4874.942,Y -1181.101,Z 999.474,A 88.44949,B 0.00000,C 180.00000} ; outside
  LIN {X 4874.942,Y -1181.101,Z 60.229,A 88.44949,B 0.00000,C 180.00000} ; preinsert
  LIN {X 4874.942,Y -1181.101,Z -189.771,A 88.44949,B 0.00000,C 180.00000} ; insert
  LIN {X 4874.942,Y -1181.101,Z -189.771,A 88.44949,B 0.00000,C 180.00000} ; release
  LIN {X 4874.942,Y -1181.101,Z 110.229,A 88.44949,B 0.00000,C 180.00000} ; retreat
  ; Step 1103, bar 2819
  LIN {X 5624.942,Y -1181.101,Z 999.474,A 88.44949,B 0.00000,C 180.00000} ; outside
  LIN {X 5624.942,Y -1181.101,Z 60.229,A 88.44949,B 0.00000,C 180.00000} ; preinsert
  LIN {X 5624.942,Y -1181.101,Z -189.771,A 88.44949,B 0.00000,C 180.00000} ; insert
  LIN {X 5624.942,Y -1181.101,Z -189.771,A 88.44949,B 0.00000,C 180.00000} ; release
  LIN {X 5624.942,Y -1181.101,Z 110.229,A 88.44949,B 0.00000,C 180.00000} ; retreat
  ; Step 1104, bar 2822
  LIN {X 6374.942,Y -1181.101,Z 999.474,A 88.44949,B 0.00000,C 180.00000} ; outside
  LIN {X 6374.942,Y -1181.101,Z 60.229,A 88.44949,B 0.00000,C 180.00000} ; preinsert
  LIN {X 6374.942,Y -1181.101,Z -189.771,A 88.44949,B 0.00000,C 180.00000} ; insert
  LIN {X 6374.942,Y -1181.101,Z -189.771,A 88.44949,B 0.00000,C 180.00000} ; release
  LIN {X 6374.942,Y -1181.101,Z 110.229,A 88.44949,B 0.00000,C 180.00000} ; retreat
  ; Step 1105, bar 2825
  LIN {X 7124.942,Y -1181.101,Z 999.474,A 88.44949,B 0.00000,C 180.00000} ; outside
  LIN {X 7124.942,Y -1181.101,Z 60.229,A 88.44949,B 0.00000,C 180.00000} ; preinsert
  LIN {X 7124.942,Y -1181.101,Z -189.771,A 88.44949,B 0.00000,C 180.00000} ; insert
  LIN {X 7124.942,Y -1181.101,Z -189.771,A 88.44949,B 0.00000,C 180.00000} ; release
  LIN {X 7124.942,Y -1181.101,Z 110.229,A 88.44949,B 0.00000,C 180.00000} ; retreat
  ; Step 1106, bar 2828
  LIN {X 7874.942,Y -1181.101,Z 999.474,A 88.44949,B 0.00000,C 180.00000} ; outside
  LIN {X 7874.942,Y -1181.101,Z 60.229,A 88.44949,B 0.00000,C 180.00000} ; preinsert
  LIN {X 7874.942,Y -1181.101,Z -189.771,A 88.44949,B 0.00000,C 180.00000} ; insert
  LIN {X 7874.942,Y -1181.101,Z -189.771,A 88.44949,B 0.00000,C 180.00000} ; release
  LIN {X 7874.942,Y -1181.101,Z 110.229,A 88.44949,B 0.00000,C 180.00000} ; retreat
  ; Step 1107, bar 2831
  LIN {X 8624.942,Y -1181.101,Z 999.474,A 88.44949,B 0.00000,C 180.00000} ; outside
  LIN {X 8624.942,Y -1181.101,Z 60.229,A 88.44949,B 0.00000,C 180.00000} ; preinsert
  LIN {X 8624.942,Y -1181.101,Z -189.771,A 88.44949,B 0.00000,C 180.00000} ; insert
  LIN {X 8624.942,Y -1181.101,Z -189.771,A 88.44949,B 0.00000,C 180.00000} ; release
  LIN {X 8624.942,Y -1181.101,Z 110.229,A 88.44949,B 0.00000,C 180.00000} ; retreat
  ; Step 1108, bar 2834
  LIN {X 9374.942,Y -1181.101,Z 999.474,A 88.44949,B 0.00000,C 180.00000} ; outside
  LIN {X 9374.942,Y -1181.101,Z 60.229,A 88.44949,B 0.00000,C 180.00000} ; preinsert
  LIN {X 9374.942,Y -1181.101,Z -189.771,A 88.44949,B 0.00000,C 180.00000} ; insert
  LIN {X 9374.942,Y -1181.101,Z -189.771,A 88.44949,B 0.00000,C 180.00000} ; release
  LIN {X 9374.942,Y -1181.101,Z 110.229,A 88.44949,B 0.00000,C 180.00000} ; retreat
  ; Step 1109, bar 2837
  LIN {X 10124.942,Y -1181.101,Z 999.474,A 88.44949,B 0.00000,C 180.00000} ; outside
  LIN {X 10124.942,Y -1181.101,Z 60.229,A 88.44949,B 0.00000,C 180.00000} ; preinsert
  LIN {X 10124.942,Y -1181.101,Z -189.771,A 88.44949,B 0.00000,C 180.00000} ; insert
  LIN {X 10124.942,Y -1181.101,Z -189.771,A 88.44949,B 0.00000,C 180.00000} ; release
  LIN {X 10124.942,Y -1181.101,Z 110.229,A 88.44949,B 0.00000,C 180.00000} ; retreat
  ; Step 1110, bar 2840
  LIN {X 10874.942,Y -1181.101,Z 999.474,A 88.44949,B 0.00000,C 180.00000} ; outside
  LIN {X 10874.942,Y -1181.101,Z 60.229,A 88.44949,B 0.00000,C 180.00000} ; preinsert
  LIN {X 10874.942,Y -1181.101,Z -189.771,A 88.44949,B 0.00000,C 180.00000} ; insert
  LIN {X 10874.942,Y -1181.101,Z -189.771,A 88.44949,B 0.00000,C 180.00000} ; release
  LIN {X 10874.942,Y -1181.101,Z 110.229,A 88.44949,B 0.00000,C 180.00000} ; retreat
  ; Step 1111, bar 2843
  LIN {X 11624.942,Y -1181.101,Z 999.474,A 88.44949,B 0.00000,C 180.00000} ; outside
  LIN {X 11624.942,Y -1181.101,Z 60.229,A 88.44949,B 0.00000,C 180.00000} ; preinsert
  LIN {X 11624.942,Y -1181.101,Z -189.771,A 88.44949,B 0.00000,C 180.00000} ; insert
  LIN {X 11624.942,Y -1181.101,Z -189.771,A 88.44949,B 0.00000,C 180.00000} ; release
  LIN {X 11624.942,Y -1181.101,Z 110.229,A 88.44949,B 0.00000,C 180.00000} ; retreat
  ; Step 1112, bar 2627
  LIN {X -11624.942,Y 1181.101,Z 999.474,A -91.55051,B 0.00000,C -180.00000} ; outside
  LIN {X -11624.942,Y 1181.101,Z 60.229,A -91.55051,B 0.00000,C -180.00000} ; preinsert
  LIN {X -11624.942,Y 1181.101,Z -189.771,A -91.55051,B 0.00000,C -180.00000} ; insert
  LIN {X -11624.942,Y 1181.101,Z -189.771,A -91.55051,B 0.00000,C -180.00000} ; release
  LIN {X -11624.942,Y 1181.101,Z 110.229,A -91.55051,B 0.00000,C -180.00000} ; retreat
  ; Step 1113, bar 2620
  LIN {X -10874.942,Y 1181.101,Z 999.474,A -91.55051,B 0.00000,C -180.00000} ; outside
  LIN {X -10874.942,Y 1181.101,Z 60.229,A -91.55051,B 0.00000,C -180.00000} ; preinsert
  LIN {X -10874.942,Y 1181.101,Z -189.771,A -91.55051,B 0.00000,C -180.00000} ; insert
  LIN {X -10874.942,Y 1181.101,Z -189.771,A -91.55051,B 0.00000,C -180.00000} ; release
  LIN {X -10874.942,Y 1181.101,Z 110.229,A -91.55051,B 0.00000,C -180.00000} ; retreat
  ; Step 1114, bar 2613
  LIN {X -10124.942,Y 1181.101,Z 999.474,A -91.55051,B 0.00000,C -180.00000} ; outside
  LIN {X -10124.942,Y 1181.101,Z 60.229,A -91.55051,B 0.00000,C -180.00000} ; preinsert
  LIN {X -10124.942,Y 1181.101,Z -189.771,A -91.55051,B 0.00000,C -180.00000} ; insert
  LIN {X -10124.942,Y 1181.101,Z -189.771,A -91.55051,B 0.00000,C -180.00000} ; release
  LIN {X -10124.942,Y 1181.101,Z 110.229,A -91.55051,B 0.00000,C -180.00000} ; retreat
  ; Step 1115, bar 2606
  LIN {X -9374.942,Y 1181.101,Z 999.474,A -91.55051,B 0.00000,C -180.00000} ; outside
  LIN {X -9374.942,Y 1181.101,Z 60.229,A -91.55051,B 0.00000,C -180.00000} ; preinsert
  LIN {X -9374.942,Y 1181.101,Z -189.771,A -91.55051,B 0.00000,C -180.00000} ; insert
  LIN {X -9374.942,Y 1181.101,Z -189.771,A -91.55051,B 0.00000,C -180.00000} ; release
  LIN {X -9374.942,Y 1181.101,Z 110.229,A -91.55051,B 0.00000,C -180.00000} ; retreat
  ; Step 1116, bar 2599
  LIN {X -8624.942,Y 1181.101,Z 999.474,A -91.55051,B 0.00000,C -180.00000} ; outside
  LIN {X -8624.942,Y 1181.101,Z 60.229,A -91.55051,B 0.00000,C -180.00000} ; preinsert
  LIN {X -8624.942,Y 1181.101,Z -189.771,A -91.55051,B 0.00000,C -180.00000} ; insert
  LIN {X -8624.942,Y 1181.101,Z -189.771,A -91.55051,B 0.00000,C -180.00000} ; release
  LIN {X -8624.942,Y 1181.101,Z 110.229,A -91.55051,B 0.00000,C -180.00000} ; retreat
  ; Step 1117, bar 2592
  LIN {X -7874.942,Y 1181.101,Z 999.474,A -91.55051,B 0.00000,C -180.00000} ; outside
  LIN {X -7874.942,Y 1181.101,Z 60.229,A -91.55051,B 0.00000,C -180.00000} ; preinsert
  LIN {X -7874.942,Y 1181.101,Z -189.771,A -91.55051,B 0.00000,C -180.00000} ; insert
  LIN {X -7874.942,Y 1181.101,Z -189.771,A -91.55051,B 0.00000,C -180.00000} ; release
  LIN {X -7874.942,Y 1181.101,Z 110.229,A -91.55051,B 0.00000,C -180.00000} ; retreat
  ; Step 1118, bar 2585
  LIN {X -7124.942,Y 1181.101,Z 999.474,A -91.55051,B 0.00000,C -180.00000} ; outside
  LIN {X -7124.942,Y 1181.101,Z 60.229,A -91.55051,B 0.00000,C -180.00000} ; preinsert
  LIN {X -7124.942,Y 1181.101,Z -189.771,A -91.55051,B 0.00000,C -180.00000} ; insert
  LIN {X -7124.942,Y 1181.101,Z -189.771,A -91.55051,B 0.00000,C -180.00000} ; release
  LIN {X -7124.942,Y 1181.101,Z 110.229,A -91.55051,B 0.00000,C -180.00000} ; retreat
  ; Step 1119, bar 2578
  LIN {X -6374.942,Y 1181.101,Z 999.474,A -91.55051,B 0.00000,C -180.00000} ; outside
  LIN {X -6374.942,Y 1181.101,Z 60.229,A -91.55051,B 0.00000,C -180.00000} ; preinsert
  LIN {X -6374.942,Y 1181.101,Z -189.771,A -91.55051,B 0.00000,C -180.00000} ; insert
  LIN {X -6374.942,Y 1181.101,Z -189.771,A -91.55051,B 0.00000,C -180.00000} ; release
  LIN {X -6374.942,Y 1181.101,Z 110.229,A -91.55051,B 0.00000,C -180.00000} ; retreat
  ; Step 1120, bar 2571
  LIN {X -5624.942,Y 1181.101,Z 999.474,A -91.55051,B 0.00000,C -180.00000} ; outside
  LIN {X -5624.942,Y 1181.101,Z 60.229,A -91.55051,B 0.00000,C -180.00000} ; preinsert
  LIN {X -5624.942,Y 1181.101,Z -189.771,A -91.55051,B 0.00000,C -180.00000} ; insert
  LIN {X -5624.942,Y 1181.101,Z -189.771,A -91.55051,B 0.00000,C -180.00000} ; release
  LIN {X -5624.942,Y 1181.101,Z 110.229,A -91.55051,B 0.00000,C -180.00000} ; retreat
  ; Step 1121, bar 2564
  LIN {X -4874.942,Y 1181.101,Z 999.474,A -91.55051,B 0.00000,C -180.00000} ; outside
  LIN {X -4874.942,Y 1181.101,Z 60.229,A -91.55051,B 0.00000,C -180.00000} ; preinsert
  LIN {X -4874.942,Y 1181.101,Z -189.771,A -91.55051,B 0.00000,C -180.00000} ; insert
  LIN {X -4874.942,Y 1181.101,Z -189.771,A -91.55051,B 0.00000,C -180.00000} ; release
  LIN {X -4874.942,Y 1181.101,Z 110.229,A -91.55051,B 0.00000,C -180.00000} ; retreat
  ; Step 1122, bar 2557
  LIN {X -4124.942,Y 1181.101,Z 999.474,A -91.55051,B 0.00000,C -180.00000} ; outside
  LIN {X -4124.942,Y 1181.101,Z 60.229,A -91.55051,B 0.00000,C -180.00000} ; preinsert
  LIN {X -4124.942,Y 1181.101,Z -189.771,A -91.55051,B 0.00000,C -180.00000} ; insert
  LIN {X -4124.942,Y 1181.101,Z -189.771,A -91.55051,B 0.00000,C -180.00000} ; release
  LIN {X -4124.942,Y 1181.101,Z 110.229,A -91.55051,B 0.00000,C -180.00000} ; retreat
  ; Step 1123, bar 2550
  LIN {X -3374.942,Y 1181.101,Z 999.474,A -91.55051,B 0.00000,C -180.00000} ; outside
  LIN {X -3374.942,Y 1181.101,Z 60.229,A -91.55051,B 0.00000,C -180.00000} ; preinsert
  LIN {X -3374.942,Y 1181.101,Z -189.771,A -91.55051,B 0.00000,C -180.00000} ; insert
  LIN {X -3374.942,Y 1181.101,Z -189.771,A -91.55051,B 0.00000,C -180.00000} ; release
  LIN {X -3374.942,Y 1181.101,Z 110.229,A -91.55051,B 0.00000,C -180.00000} ; retreat
  ; Step 1124, bar 2543
  LIN {X -2624.942,Y 1181.101,Z 999.474,A -91.55051,B 0.00000,C -180.00000} ; outside
  LIN {X -2624.942,Y 1181.101,Z 60.229,A -91.55051,B 0.00000,C -180.00000} ; preinsert
  LIN {X -2624.942,Y 1181.101,Z -189.771,A -91.55051,B 0.00000,C -180.00000} ; insert
  LIN {X -2624.942,Y 1181.101,Z -189.771,A -91.55051,B 0.00000,C -180.00000} ; release
  LIN {X -2624.942,Y 1181.101,Z 110.229,A -91.55051,B 0.00000,C -180.00000} ; retreat
  ; Step 1125, bar 2536
  LIN {X -1874.942,Y 1181.101,Z 999.474,A -91.55051,B 0.00000,C -180.00000} ; outside
  LIN {X -1874.942,Y 1181.101,Z 60.229,A -91.55051,B 0.00000,C -180.00000} ; preinsert
  LIN {X -1874.942,Y 1181.101,Z -189.771,A -91.55051,B 0.00000,C -180.00000} ; insert
  LIN {X -1874.942,Y 1181.101,Z -189.771,A -91.55051,B 0.00000,C -180.00000} ; release
  LIN {X -1874.942,Y 1181.101,Z 110.229,A -91.55051,B 0.00000,C -180.00000} ; retreat
  ; Step 1126, bar 2529
  LIN {X -1124.942,Y 1181.101,Z 999.474,A -91.55051,B 0.00000,C -180.00000} ; outside
  LIN {X -1124.942,Y 1181.101,Z 60.229,A -91.55051,B 0.00000,C -180.00000} ; preinsert
  LIN {X -1124.942,Y 1181.101,Z -189.771,A -91.55051,B 0.00000,C -180.00000} ; insert
  LIN {X -1124.942,Y 1181.101,Z -189.771,A -91.55051,B 0.00000,C -180.00000} ; release
  LIN {X -1124.942,Y 1181.101,Z 110.229,A -91.55051,B 0.00000,C -180.00000} ; retreat
  ; Step 1127, bar 1970
  LIN {X -374.942,Y 1181.101,Z 999.474,A -91.55051,B 0.00000,C 180.00000} ; outside
  LIN {X -374.942,Y 1181.101,Z 60.229,A -91.55051,B 0.00000,C 180.00000} ; preinsert
  LIN {X -374.942,Y 1181.101,Z -189.771,A -91.55051,B 0.00000,C 180.00000} ; insert
  LIN {X -374.942,Y 1181.101,Z -189.771,A -91.55051,B 0.00000,C 180.00000} ; release
  LIN {X -374.942,Y 1181.101,Z 110.229,A -91.55051,B 0.00000,C 180.00000} ; retreat
  ; Step 1128, bar 280
  LIN {X 0.000,Y -250.000,Z 1128.121,A 0.00000,B 0.00000,C 180.00000} ; outside
  LIN {X 0.000,Y -250.000,Z 188.371,A 0.00000,B 0.00000,C 180.00000} ; preinsert
  LIN {X 0.000,Y -250.000,Z -61.629,A 0.00000,B 0.00000,C 180.00000} ; insert
  LIN {X 0.000,Y -250.000,Z -61.629,A 0.00000,B 0.00000,C 180.00000} ; release
  LIN {X 0.000,Y -250.000,Z 238.371,A 0.00000,B 0.00000,C 180.00000} ; retreat
  ; Step 1129, bar 307
  LIN {X 0.000,Y 250.000,Z 1128.121,A 0.00000,B 0.00000,C 180.00000} ; outside
  LIN {X 0.000,Y 250.000,Z 188.371,A 0.00000,B 0.00000,C 180.00000} ; preinsert
  LIN {X 0.000,Y 250.000,Z -61.629,A 0.00000,B 0.00000,C 180.00000} ; insert
  LIN {X 0.000,Y 250.000,Z -61.629,A 0.00000,B 0.00000,C 180.00000} ; release
  LIN {X 0.000,Y 250.000,Z 238.371,A 0.00000,B 0.00000,C 180.00000} ; retreat
  ; Step 1130, bar 1480
  LIN {X 14334.988,Y 2494.793,Z 907.454,A -89.99654,B 0.00000,C 180.00000} ; outside
  LIN {X 14334.988,Y 2494.793,Z -78.660,A -89.99654,B 0.00000,C 180.00000} ; preinsert
